(* CODESYS project TouchPanel-PIO3_MB_EC.ecp

Project tree, tasks and I/O mapping:
  TP_EtherCat : TP600 10.1 1280x800 PIO3 CP , WAGO, order no. 0762-5304, version 5.13.2.32
    application Application
      libraries: ; VisuDialogs, * (System); SysFile23, 3.5.13.0 (System); VisuElemBase, 3.5.13.20 (System); SysPlcCtrl23, 3.5.13.0 (System); SysTime, 3.5.9.0 (System)
      task PLC_Task (cyclic, interval t#10ms, priority 13) calls nothing
      task EtherCAT_Task (cyclic, interval 4 ms, priority 6) calls PLC_PRG
      program PLC_PRG [ST]
      data type typDiagnosticStatusWord
      data type typDSW
      data type typEcDiag
      function block fbSdoRead4 [ST]
      function block fbSdoWrite [ST]
      program prgSdoHandling [ST]
    Serial
      COM1 : COM1, WAGO, version 0.0.0.19
    MODBUS
      MODBUS : MODBUS, WAGO, order no. n/a, version 1.1.1.15
        _internal_1006_0001_Master : MODBUS Master, WAGO, order no. n/a, version 1.1.1.15
    CANbus
    e_Display_Onboard_IO : TP600 Onboard IO, WAGO, version 0.0.1.2
        unmapped channels: _IN, _OUT
    EtherCAT_Master : EtherCAT Master, WAGO, version 3.5.13.21
        settings: NetworkName = 'ethX2'; NetworkName = "ethX2"; SelectNetworkByName = TRUE
      _750_354_000_002_EtherCat_fieldbus_coupler : 750-354/000-002 EtherCat fieldbus coupler, WAGO, order no. 750-354/000-002, version Revision=16#10010002
          settings: ModularDevice = True; MDP_InputOffsets = [0,224,0,32,96,160]; MDP_OutputOffsets = [0,0,224,32,96,160]; Physical Address of the Slave = 1001; Sync.Length = 30; Sync.Length = 30; FMMU.Global Start Address = 16#02000000; FMMU.Length = 30; FMMU.Physical Start Address = 16#1800; FMMU.Access = 16#02; FMMU.Global Start Address = 16#01000000; FMMU.Length = 30; FMMU.Physical Start Address = 16#2400; FMMU.Access = 16#01; FMMU.Global Start Address = 16#00080000; FMMU.Physical Start Address = 16#080D; FMMU.Access = 16#01; Number of RxPDOs of the Slave = 5; Number of TxPDOs of the Slave = 5; DC sync0 cycletime = 4000; DC sync1 cycletime = 4000; Number of SDO = 1; Explicit Device ID (Upper 8 bits).Index = 16#2134; Explicit Device ID (Upper 8 bits).Subindex = 16#00; Explicit Device ID (Upper 8 bits).Value = 0; Explicit Device ID (Upper 8 bits).Size = 8; Explicit Device ID (Upper 8 bits).AbortIfError = FALSE; Explicit Device ID (Upper 8 bits).JumpToLine = FALSE; Explicit Device ID (Upper 8 bits).Line = 0; Explicit Device ID (Upper 8 bits).CompleteAccess = False; RxTxPdo.NumberofExcludes = 0; RxTxPdo.NumberofEntries = 6; RxTxPdo.Index = 16#16FF; RxTxPdo.Fixed = True; RxTxPdo.Mandatory = True; RxTxPdo.Virtual = False; RxTxPdo.Sm = 2; RxTxPdo.Su = 2; RxTxPdo.Name = 'Output'; RxTxPdo.DependOnSlot = False;
            RxTxPdo.DependOnSlotGroup = False; RxTxPdo.OverwrittenByModule = False; FC Control, K-Bus Cycle Overrun Flag Disable.Index = 16#F200; FC Control, K-Bus Cycle Overrun Flag Disable.SubIndex = 1; FC Control, K-Bus Cycle Overrun Flag Disable.Size = 1; FC Control, K-Bus Cycle Overrun Flag Disable.Offset = 0; FC Control, K-Bus Cycle Overrun Flag Disable.DependOnSlot = False; FC Control, K-Bus Cycle Overrun Flag Disable.DependOnSlotGroup = False; FC Control, Input Process Data Hold Request.Index = 16#F200; FC Control, Input Process Data Hold Request.SubIndex = 2; FC Control, Input Process Data Hold Request.Size = 1; FC Control, Input Process Data Hold Request.Offset = 0; FC Control, Input Process Data Hold Request.DependOnSlot = False; FC Control, Input Process Data Hold Request.DependOnSlotGroup = False; FC Control, Output Process Data Hold Request.Index = 16#F200; FC Control, Output Process Data Hold Request.SubIndex = 3; FC Control, Output Process Data Hold Request.Size = 1; FC Control, Output Process Data Hold Request.Offset = 0; FC Control, Output Process Data Hold Request.DependOnSlot = False; FC Control, Output Process Data Hold Request.DependOnSlotGroup = False; FC Control, Output Process Data Clear Request.Index = 16#F200; FC Control, Output Process Data Clear Request.SubIndex = 4; FC Control, Output Process Data Clear Request.Size = 1; FC Control, Output Process Data Clear Request.Offset = 0; FC Control, Output Process Data Clear Request.DependOnSlot = False; FC Control, Output Process Data Clear Request.DependOnSlotGroup = False; Entry.Index = 16#0000; Entry.SubIndex = 0; Entry.Size = 12; Entry.Offset = 0; Entry.DependOnSlot = False; Entry.DependOnSlotGroup = False; Diagnostics Control Word.Index = 16#F200; Diagnostics Control Word.SubIndex = 5; Diagnostics Control Word.Size = 16; Diagnostics Control Word.Offset = 0; Diagnostics Control Word.DependOnSlot = False; Diagnostics Control Word.DependOnSlotGroup = False; RxTxPdo.NumberofExcludes = 0; RxTxPdo.NumberofEntries = 6;
            RxTxPdo.Index = 16#1602; RxTxPdo.Fixed = True; RxTxPdo.Mandatory = True; RxTxPdo.Virtual = False; RxTxPdo.Sm = 2; RxTxPdo.Su = 0; RxTxPdo.Name = 'Output(s)'; RxTxPdo.DependOnSlot = True; RxTxPdo.DependOnSlotGroup = False; RxTxPdo.OverwrittenByModule = True; Channel 1, Control.Index = 16#7020; Channel 1, Control.SubIndex = 1; Channel 1, Control.Size = 8; Channel 1, Control.Offset = 0; Channel 1, Control.DependOnSlot = True; Channel 1, Control.DependOnSlotGroup = True; ---.Index = 16#0000; ---.SubIndex = 0; ---.Size = 8; ---.Offset = 0; ---.DependOnSlot = False; ---.DependOnSlotGroup = False; Channel 1, Word 1.Index = 16#7020; Channel 1, Word 1.SubIndex = 2; Channel 1, Word 1.Size = 16; Channel 1, Word 1.Offset = 0; Channel 1, Word 1.DependOnSlot = True; Channel 1, Word 1.DependOnSlotGroup = True; Channel 2, Control.Index = 16#7020; Channel 2, Control.SubIndex = 3; Channel 2, Control.Size = 8; Channel 2, Control.Offset = 0; Channel 2, Control.DependOnSlot = True; Channel 2, Control.DependOnSlotGroup = True; ---.Index = 16#0000; ---.SubIndex = 0; ---.Size = 8; ---.Offset = 0; ---.DependOnSlot = False; ---.DependOnSlotGroup = False;
            Channel 2, Word 1.Index = 16#7020; Channel 2, Word 1.SubIndex = 4; Channel 2, Word 1.Size = 16; Channel 2, Word 1.Offset = 0; Channel 2, Word 1.DependOnSlot = True; Channel 2, Word 1.DependOnSlotGroup = True; RxTxPdo.NumberofExcludes = 0; RxTxPdo.NumberofEntries = 6; RxTxPdo.Index = 16#1603; RxTxPdo.Fixed = True; RxTxPdo.Mandatory = True; RxTxPdo.Virtual = False; RxTxPdo.Sm = 2; RxTxPdo.Su = 0; RxTxPdo.Name = 'Output(s)'; RxTxPdo.DependOnSlot = True; RxTxPdo.DependOnSlotGroup = False; RxTxPdo.OverwrittenByModule = True; Channel 1, Control.Index = 16#7030; Channel 1, Control.SubIndex = 1; Channel 1, Control.Size = 8; Channel 1, Control.Offset = 0; Channel 1, Control.DependOnSlot = True; Channel 1, Control.DependOnSlotGroup = True; ---.Index = 16#0000; ---.SubIndex = 0; ---.Size = 8; ---.Offset = 0; ---.DependOnSlot = False; ---.DependOnSlotGroup = False; Channel 1, Word 1.Index = 16#7030; Channel 1, Word 1.SubIndex = 2; Channel 1, Word 1.Size = 16; Channel 1, Word 1.Offset = 0; Channel 1, Word 1.DependOnSlot = True; Channel 1, Word 1.DependOnSlotGroup = True; Channel 2, Control.Index = 16#7030; Channel 2, Control.SubIndex = 3; Channel 2, Control.Size = 8; Channel 2, Control.Offset = 0;
            Channel 2, Control.DependOnSlot = True; Channel 2, Control.DependOnSlotGroup = True; ---.Index = 16#0000; ---.SubIndex = 0; ---.Size = 8; ---.Offset = 0; ---.DependOnSlot = False; ---.DependOnSlotGroup = False; Channel 2, Word 1.Index = 16#7030; Channel 2, Word 1.SubIndex = 4; Channel 2, Word 1.Size = 16; Channel 2, Word 1.Offset = 0; Channel 2, Word 1.DependOnSlot = True; Channel 2, Word 1.DependOnSlotGroup = True; RxTxPdo.NumberofExcludes = 0; RxTxPdo.NumberofEntries = 6; RxTxPdo.Index = 16#1604; RxTxPdo.Fixed = True; RxTxPdo.Mandatory = True; RxTxPdo.Virtual = False; RxTxPdo.Sm = 2; RxTxPdo.Su = 0; RxTxPdo.Name = 'Output(s)'; RxTxPdo.DependOnSlot = True; RxTxPdo.DependOnSlotGroup = False; RxTxPdo.OverwrittenByModule = True; Channel 1, Control.Index = 16#7040; Channel 1, Control.SubIndex = 1; Channel 1, Control.Size = 8; Channel 1, Control.Offset = 0; Channel 1, Control.DependOnSlot = True; Channel 1, Control.DependOnSlotGroup = True; ---.Index = 16#0000; ---.SubIndex = 0; ---.Size = 8; ---.Offset = 0; ---.DependOnSlot = False; ---.DependOnSlotGroup = False; Channel 1, Word 1.Index = 16#7040; Channel 1, Word 1.SubIndex = 2;
            Channel 1, Word 1.Size = 16; Channel 1, Word 1.Offset = 0; Channel 1, Word 1.DependOnSlot = True; Channel 1, Word 1.DependOnSlotGroup = True; Channel 2, Control.Index = 16#7040; Channel 2, Control.SubIndex = 3; Channel 2, Control.Size = 8; Channel 2, Control.Offset = 0; Channel 2, Control.DependOnSlot = True; Channel 2, Control.DependOnSlotGroup = True; ---.Index = 16#0000; ---.SubIndex = 0; ---.Size = 8; ---.Offset = 0; ---.DependOnSlot = False; ---.DependOnSlotGroup = False; Channel 2, Word 1.Index = 16#7040; Channel 2, Word 1.SubIndex = 4; Channel 2, Word 1.Size = 16; Channel 2, Word 1.Offset = 0; Channel 2, Word 1.DependOnSlot = True; Channel 2, Word 1.DependOnSlotGroup = True; RxTxPdo.NumberofExcludes = 0; RxTxPdo.NumberofEntries = 16; RxTxPdo.Index = 16#1601; RxTxPdo.Fixed = True; RxTxPdo.Mandatory = True; RxTxPdo.Virtual = False; RxTxPdo.Sm = 2; RxTxPdo.Su = 0; RxTxPdo.Name = 'Output(s)'; RxTxPdo.DependOnSlot = True; RxTxPdo.DependOnSlotGroup = False; RxTxPdo.OverwrittenByModule = True; Channel 1, Data 1.Index = 16#7010; Channel 1, Data 1.SubIndex = 1; Channel 1, Data 1.Size = 1; Channel 1, Data 1.Offset = 0; Channel 1, Data 1.DependOnSlot = True; Channel 1, Data 1.DependOnSlotGroup = True;
            Channel 2, Data 1.Index = 16#7010; Channel 2, Data 1.SubIndex = 2; Channel 2, Data 1.Size = 1; Channel 2, Data 1.Offset = 0; Channel 2, Data 1.DependOnSlot = True; Channel 2, Data 1.DependOnSlotGroup = True; Channel 3, Data 1.Index = 16#7010; Channel 3, Data 1.SubIndex = 3; Channel 3, Data 1.Size = 1; Channel 3, Data 1.Offset = 0; Channel 3, Data 1.DependOnSlot = True; Channel 3, Data 1.DependOnSlotGroup = True; Channel 4, Data 1.Index = 16#7010; Channel 4, Data 1.SubIndex = 4; Channel 4, Data 1.Size = 1; Channel 4, Data 1.Offset = 0; Channel 4, Data 1.DependOnSlot = True; Channel 4, Data 1.DependOnSlotGroup = True; Channel 5, Data 1.Index = 16#7010; Channel 5, Data 1.SubIndex = 5; Channel 5, Data 1.Size = 1; Channel 5, Data 1.Offset = 0; Channel 5, Data 1.DependOnSlot = True; Channel 5, Data 1.DependOnSlotGroup = True; Channel 6, Data 1.Index = 16#7010; Channel 6, Data 1.SubIndex = 6; Channel 6, Data 1.Size = 1; Channel 6, Data 1.Offset = 0; Channel 6, Data 1.DependOnSlot = True; Channel 6, Data 1.DependOnSlotGroup = True; Channel 7, Data 1.Index = 16#7010; Channel 7, Data 1.SubIndex = 7; Channel 7, Data 1.Size = 1; Channel 7, Data 1.Offset = 0; Channel 7, Data 1.DependOnSlot = True; Channel 7, Data 1.DependOnSlotGroup = True; Channel 8, Data 1.Index = 16#7010; Channel 8, Data 1.SubIndex = 8; Channel 8, Data 1.Size = 1; Channel 8, Data 1.Offset = 0;
            Channel 8, Data 1.DependOnSlot = True; Channel 8, Data 1.DependOnSlotGroup = True; Channel 9, Data 1.Index = 16#7010; Channel 9, Data 1.SubIndex = 9; Channel 9, Data 1.Size = 1; Channel 9, Data 1.Offset = 0; Channel 9, Data 1.DependOnSlot = True; Channel 9, Data 1.DependOnSlotGroup = True; Channel 10, Data 1.Index = 16#7010; Channel 10, Data 1.SubIndex = 10; Channel 10, Data 1.Size = 1; Channel 10, Data 1.Offset = 0; Channel 10, Data 1.DependOnSlot = True; Channel 10, Data 1.DependOnSlotGroup = True; Channel 11, Data 1.Index = 16#7010; Channel 11, Data 1.SubIndex = 11; Channel 11, Data 1.Size = 1; Channel 11, Data 1.Offset = 0; Channel 11, Data 1.DependOnSlot = True; Channel 11, Data 1.DependOnSlotGroup = True; Channel 12, Data 1.Index = 16#7010; Channel 12, Data 1.SubIndex = 12; Channel 12, Data 1.Size = 1; Channel 12, Data 1.Offset = 0; Channel 12, Data 1.DependOnSlot = True; Channel 12, Data 1.DependOnSlotGroup = True; Channel 13, Data 1.Index = 16#7010; Channel 13, Data 1.SubIndex = 13; Channel 13, Data 1.Size = 1; Channel 13, Data 1.Offset = 0; Channel 13, Data 1.DependOnSlot = True; Channel 13, Data 1.DependOnSlotGroup = True; Channel 14, Data 1.Index = 16#7010; Channel 14, Data 1.SubIndex = 14; Channel 14, Data 1.Size = 1; Channel 14, Data 1.Offset = 0; Channel 14, Data 1.DependOnSlot = True; Channel 14, Data 1.DependOnSlotGroup = True; Channel 15, Data 1.Index = 16#7010; Channel 15, Data 1.SubIndex = 15;
            Channel 15, Data 1.Size = 1; Channel 15, Data 1.Offset = 0; Channel 15, Data 1.DependOnSlot = True; Channel 15, Data 1.DependOnSlotGroup = True; Channel 16, Data 1.Index = 16#7010; Channel 16, Data 1.SubIndex = 16; Channel 16, Data 1.Size = 1; Channel 16, Data 1.Offset = 0; Channel 16, Data 1.DependOnSlot = True; Channel 16, Data 1.DependOnSlotGroup = True; RxTxPdo.NumberofExcludes = 0; RxTxPdo.NumberofEntries = 7; RxTxPdo.Index = 16#1AFF; RxTxPdo.Fixed = True; RxTxPdo.Mandatory = True; RxTxPdo.Virtual = False; RxTxPdo.Sm = 3; RxTxPdo.Su = 3; RxTxPdo.Name = 'Input'; RxTxPdo.DependOnSlot = False; RxTxPdo.DependOnSlotGroup = False; RxTxPdo.OverwrittenByModule = False; FC Status, K-Bus Cycle Overrun Flag.Index = 16#F100; FC Status, K-Bus Cycle Overrun Flag.SubIndex = 1; FC Status, K-Bus Cycle Overrun Flag.Size = 1; FC Status, K-Bus Cycle Overrun Flag.Offset = 0; FC Status, K-Bus Cycle Overrun Flag.DependOnSlot = False; FC Status, K-Bus Cycle Overrun Flag.DependOnSlotGroup = False; FC Status, Input Process Data Hold Ack..Index = 16#F100; FC Status, Input Process Data Hold Ack..SubIndex = 2; FC Status, Input Process Data Hold Ack..Size = 1; FC Status, Input Process Data Hold Ack..Offset = 0; FC Status, Input Process Data Hold Ack..DependOnSlot = False; FC Status, Input Process Data Hold Ack..DependOnSlotGroup = False; FC Status, Output Process Data Hold Ack..Index = 16#F100; FC Status, Output Process Data Hold Ack..SubIndex = 3; FC Status, Output Process Data Hold Ack..Size = 1; FC Status, Output Process Data Hold Ack..Offset = 0; FC Status, Output Process Data Hold Ack..DependOnSlot = False; FC Status, Output Process Data Hold Ack..DependOnSlotGroup = False;
            FC Status, Output Process Data Clear Ack..Index = 16#F100; FC Status, Output Process Data Clear Ack..SubIndex = 4; FC Status, Output Process Data Clear Ack..Size = 1; FC Status, Output Process Data Clear Ack..Offset = 0; FC Status, Output Process Data Clear Ack..DependOnSlot = False; FC Status, Output Process Data Clear Ack..DependOnSlotGroup = False; Entry.Index = 16#0000; Entry.SubIndex = 0; Entry.Size = 11; Entry.Offset = 0; Entry.DependOnSlot = False; Entry.DependOnSlotGroup = False; Diagnosis History, New Message Available.Index = 16#10F3; Diagnosis History, New Message Available.SubIndex = 4; Diagnosis History, New Message Available.Size = 1; Diagnosis History, New Message Available.Offset = 0; Diagnosis History, New Message Available.DependOnSlot = False; Diagnosis History, New Message Available.DependOnSlotGroup = False; Diagnostics Status Word.Index = 16#F100; Diagnostics Status Word.SubIndex = 5; Diagnostics Status Word.Size = 16; Diagnostics Status Word.Offset = 0; Diagnostics Status Word.DependOnSlot = False; Diagnostics Status Word.DependOnSlotGroup = False; RxTxPdo.NumberofExcludes = 0; RxTxPdo.NumberofEntries = 6; RxTxPdo.Index = 16#1A02; RxTxPdo.Fixed = True; RxTxPdo.Mandatory = True; RxTxPdo.Virtual = False; RxTxPdo.Sm = 3; RxTxPdo.Su = 0; RxTxPdo.Name = 'Input(s)'; RxTxPdo.DependOnSlot = True; RxTxPdo.DependOnSlotGroup = False; RxTxPdo.OverwrittenByModule = True; Channel 1, Status.Index = 16#6020; Channel 1, Status.SubIndex = 1; Channel 1, Status.Size = 8; Channel 1, Status.Offset = 0;
            Channel 1, Status.DependOnSlot = True; Channel 1, Status.DependOnSlotGroup = True; ---.Index = 16#0000; ---.SubIndex = 0; ---.Size = 8; ---.Offset = 0; ---.DependOnSlot = False; ---.DependOnSlotGroup = False; Channel 1, Word 1.Index = 16#6020; Channel 1, Word 1.SubIndex = 2; Channel 1, Word 1.Size = 16; Channel 1, Word 1.Offset = 0; Channel 1, Word 1.DependOnSlot = True; Channel 1, Word 1.DependOnSlotGroup = True; Channel 2, Status.Index = 16#6020; Channel 2, Status.SubIndex = 3; Channel 2, Status.Size = 8; Channel 2, Status.Offset = 0; Channel 2, Status.DependOnSlot = True; Channel 2, Status.DependOnSlotGroup = True; ---.Index = 16#0000; ---.SubIndex = 0; ---.Size = 8; ---.Offset = 0; ---.DependOnSlot = False; ---.DependOnSlotGroup = False; Channel 2, Word 1.Index = 16#6020; Channel 2, Word 1.SubIndex = 4; Channel 2, Word 1.Size = 16; Channel 2, Word 1.Offset = 0; Channel 2, Word 1.DependOnSlot = True; Channel 2, Word 1.DependOnSlotGroup = True; RxTxPdo.NumberofExcludes = 0; RxTxPdo.NumberofEntries = 6; RxTxPdo.Index = 16#1A03; RxTxPdo.Fixed = True; RxTxPdo.Mandatory = True; RxTxPdo.Virtual = False; RxTxPdo.Sm = 3; RxTxPdo.Su = 0;
            RxTxPdo.Name = 'Input(s)'; RxTxPdo.DependOnSlot = True; RxTxPdo.DependOnSlotGroup = False; RxTxPdo.OverwrittenByModule = True; Channel 1, Status.Index = 16#6030; Channel 1, Status.SubIndex = 1; Channel 1, Status.Size = 8; Channel 1, Status.Offset = 0; Channel 1, Status.DependOnSlot = True; Channel 1, Status.DependOnSlotGroup = True; ---.Index = 16#0000; ---.SubIndex = 0; ---.Size = 8; ---.Offset = 0; ---.DependOnSlot = False; ---.DependOnSlotGroup = False; Channel 1, Word 1.Index = 16#6030; Channel 1, Word 1.SubIndex = 2; Channel 1, Word 1.Size = 16; Channel 1, Word 1.Offset = 0; Channel 1, Word 1.DependOnSlot = True; Channel 1, Word 1.DependOnSlotGroup = True; Channel 2, Status.Index = 16#6030; Channel 2, Status.SubIndex = 3; Channel 2, Status.Size = 8; Channel 2, Status.Offset = 0; Channel 2, Status.DependOnSlot = True; Channel 2, Status.DependOnSlotGroup = True; ---.Index = 16#0000; ---.SubIndex = 0; ---.Size = 8; ---.Offset = 0; ---.DependOnSlot = False; ---.DependOnSlotGroup = False; Channel 2, Word 1.Index = 16#6030; Channel 2, Word 1.SubIndex = 4; Channel 2, Word 1.Size = 16; Channel 2, Word 1.Offset = 0; Channel 2, Word 1.DependOnSlot = True; Channel 2, Word 1.DependOnSlotGroup = True;
            RxTxPdo.NumberofExcludes = 0; RxTxPdo.NumberofEntries = 6; RxTxPdo.Index = 16#1A04; RxTxPdo.Fixed = True; RxTxPdo.Mandatory = True; RxTxPdo.Virtual = False; RxTxPdo.Sm = 3; RxTxPdo.Su = 0; RxTxPdo.Name = 'Input(s)'; RxTxPdo.DependOnSlot = True; RxTxPdo.DependOnSlotGroup = False; RxTxPdo.OverwrittenByModule = True; Channel 1, Status.Index = 16#6040; Channel 1, Status.SubIndex = 1; Channel 1, Status.Size = 8; Channel 1, Status.Offset = 0; Channel 1, Status.DependOnSlot = True; Channel 1, Status.DependOnSlotGroup = True; ---.Index = 16#0000; ---.SubIndex = 0; ---.Size = 8; ---.Offset = 0; ---.DependOnSlot = False; ---.DependOnSlotGroup = False; Channel 1, Word 1.Index = 16#6040; Channel 1, Word 1.SubIndex = 2; Channel 1, Word 1.Size = 16; Channel 1, Word 1.Offset = 0; Channel 1, Word 1.DependOnSlot = True; Channel 1, Word 1.DependOnSlotGroup = True; Channel 2, Status.Index = 16#6040; Channel 2, Status.SubIndex = 3; Channel 2, Status.Size = 8; Channel 2, Status.Offset = 0; Channel 2, Status.DependOnSlot = True; Channel 2, Status.DependOnSlotGroup = True; ---.Index = 16#0000; ---.SubIndex = 0; ---.Size = 8; ---.Offset = 0;
            ---.DependOnSlot = False; ---.DependOnSlotGroup = False; Channel 2, Word 1.Index = 16#6040; Channel 2, Word 1.SubIndex = 4; Channel 2, Word 1.Size = 16; Channel 2, Word 1.Offset = 0; Channel 2, Word 1.DependOnSlot = True; Channel 2, Word 1.DependOnSlotGroup = True; RxTxPdo.NumberofExcludes = 0; RxTxPdo.NumberofEntries = 16; RxTxPdo.Index = 16#1A00; RxTxPdo.Fixed = True; RxTxPdo.Mandatory = True; RxTxPdo.Virtual = False; RxTxPdo.Sm = 3; RxTxPdo.Su = 0; RxTxPdo.Name = 'Input(s)'; RxTxPdo.DependOnSlot = True; RxTxPdo.DependOnSlotGroup = False; RxTxPdo.OverwrittenByModule = True; Channel 1, Data 1.Index = 16#6000; Channel 1, Data 1.SubIndex = 1; Channel 1, Data 1.Size = 1; Channel 1, Data 1.Offset = 0; Channel 1, Data 1.DependOnSlot = True; Channel 1, Data 1.DependOnSlotGroup = True; Channel 2, Data 1.Index = 16#6000; Channel 2, Data 1.SubIndex = 2; Channel 2, Data 1.Size = 1; Channel 2, Data 1.Offset = 0; Channel 2, Data 1.DependOnSlot = True; Channel 2, Data 1.DependOnSlotGroup = True; Channel 3, Data 1.Index = 16#6000; Channel 3, Data 1.SubIndex = 3; Channel 3, Data 1.Size = 1; Channel 3, Data 1.Offset = 0; Channel 3, Data 1.DependOnSlot = True; Channel 3, Data 1.DependOnSlotGroup = True; Channel 4, Data 1.Index = 16#6000; Channel 4, Data 1.SubIndex = 4;
            Channel 4, Data 1.Size = 1; Channel 4, Data 1.Offset = 0; Channel 4, Data 1.DependOnSlot = True; Channel 4, Data 1.DependOnSlotGroup = True; Channel 5, Data 1.Index = 16#6000; Channel 5, Data 1.SubIndex = 5; Channel 5, Data 1.Size = 1; Channel 5, Data 1.Offset = 0; Channel 5, Data 1.DependOnSlot = True; Channel 5, Data 1.DependOnSlotGroup = True; Channel 6, Data 1.Index = 16#6000; Channel 6, Data 1.SubIndex = 6; Channel 6, Data 1.Size = 1; Channel 6, Data 1.Offset = 0; Channel 6, Data 1.DependOnSlot = True; Channel 6, Data 1.DependOnSlotGroup = True; Channel 7, Data 1.Index = 16#6000; Channel 7, Data 1.SubIndex = 7; Channel 7, Data 1.Size = 1; Channel 7, Data 1.Offset = 0; Channel 7, Data 1.DependOnSlot = True; Channel 7, Data 1.DependOnSlotGroup = True; Channel 8, Data 1.Index = 16#6000; Channel 8, Data 1.SubIndex = 8; Channel 8, Data 1.Size = 1; Channel 8, Data 1.Offset = 0; Channel 8, Data 1.DependOnSlot = True; Channel 8, Data 1.DependOnSlotGroup = True; Channel 9, Data 1.Index = 16#6000; Channel 9, Data 1.SubIndex = 9; Channel 9, Data 1.Size = 1; Channel 9, Data 1.Offset = 0; Channel 9, Data 1.DependOnSlot = True; Channel 9, Data 1.DependOnSlotGroup = True; Channel 10, Data 1.Index = 16#6000; Channel 10, Data 1.SubIndex = 10; Channel 10, Data 1.Size = 1; Channel 10, Data 1.Offset = 0; Channel 10, Data 1.DependOnSlot = True; Channel 10, Data 1.DependOnSlotGroup = True;
            Channel 11, Data 1.Index = 16#6000; Channel 11, Data 1.SubIndex = 11; Channel 11, Data 1.Size = 1; Channel 11, Data 1.Offset = 0; Channel 11, Data 1.DependOnSlot = True; Channel 11, Data 1.DependOnSlotGroup = True; Channel 12, Data 1.Index = 16#6000; Channel 12, Data 1.SubIndex = 12; Channel 12, Data 1.Size = 1; Channel 12, Data 1.Offset = 0; Channel 12, Data 1.DependOnSlot = True; Channel 12, Data 1.DependOnSlotGroup = True; Channel 13, Data 1.Index = 16#6000; Channel 13, Data 1.SubIndex = 13; Channel 13, Data 1.Size = 1; Channel 13, Data 1.Offset = 0; Channel 13, Data 1.DependOnSlot = True; Channel 13, Data 1.DependOnSlotGroup = True; Channel 14, Data 1.Index = 16#6000; Channel 14, Data 1.SubIndex = 14; Channel 14, Data 1.Size = 1; Channel 14, Data 1.Offset = 0; Channel 14, Data 1.DependOnSlot = True; Channel 14, Data 1.DependOnSlotGroup = True; Channel 15, Data 1.Index = 16#6000; Channel 15, Data 1.SubIndex = 15; Channel 15, Data 1.Size = 1; Channel 15, Data 1.Offset = 0; Channel 15, Data 1.DependOnSlot = True; Channel 15, Data 1.DependOnSlotGroup = True; Channel 16, Data 1.Index = 16#6000; Channel 16, Data 1.SubIndex = 16; Channel 16, Data 1.Size = 1; Channel 16, Data 1.Offset = 0; Channel 16, Data 1.DependOnSlot = True; Channel 16, Data 1.DependOnSlotGroup = True; FC Control, K-Bus Cycle Overrun Flag Disable.Name = 'FC Control, K-Bus Cycle Overrun Flag Disable'; FC Control, K-Bus Cycle Overrun Flag Disable.DataType = 'BIT'; FC Control, K-Bus Cycle Overrun Flag Disable.Default = ''; FC Control, K-Bus Cycle Overrun Flag Disable.Comment = '';
            FC Control, Input Process Data Hold Request.Name = 'FC Control, Input Process Data Hold Request'; FC Control, Input Process Data Hold Request.DataType = 'BIT'; FC Control, Input Process Data Hold Request.Default = ''; FC Control, Input Process Data Hold Request.Comment = ''; FC Control, Output Process Data Hold Request.Name = 'FC Control, Output Process Data Hold Request'; FC Control, Output Process Data Hold Request.DataType = 'BIT'; FC Control, Output Process Data Hold Request.Default = ''; FC Control, Output Process Data Hold Request.Comment = ''; FC Control, Output Process Data Clear Request.Name = 'FC Control, Output Process Data Clear Request'; FC Control, Output Process Data Clear Request.DataType = 'BIT'; FC Control, Output Process Data Clear Request.Default = ''; FC Control, Output Process Data Clear Request.Comment = ''; Entry.Name = ''; Entry.DataType = ''; Entry.Default = ''; Entry.Comment = ''; Diagnostics Control Word.Name = 'Diagnostics Control Word'; Diagnostics Control Word.DataType = 'UINT'; Diagnostics Control Word.Default = ''; Diagnostics Control Word.Comment = ''; Channel 1, Control.Name = 'Channel 1, Control'; Channel 1, Control.DataType = 'USINT'; Channel 1, Control.Default = ''; Channel 1, Control.Comment = ''; ---.Name = '---'; ---.DataType = ''; ---.Default = ''; ---.Comment = ''; Channel 1, Word 1.Name = 'Channel 1, Word 1'; Channel 1, Word 1.DataType = 'UINT'; Channel 1, Word 1.Default = ''; Channel 1, Word 1.Comment = ''; Channel 2, Control.Name = 'Channel 2, Control'; Channel 2, Control.DataType = 'USINT'; Channel 2, Control.Default = ''; Channel 2, Control.Comment = ''; ---.Name = '---'; ---.DataType = ''; ---.Default = ''; ---.Comment = '';
            Channel 2, Word 1.Name = 'Channel 2, Word 1'; Channel 2, Word 1.DataType = 'UINT'; Channel 2, Word 1.Default = ''; Channel 2, Word 1.Comment = ''; Channel 1, Control.Name = 'Channel 1, Control'; Channel 1, Control.DataType = 'USINT'; Channel 1, Control.Default = ''; Channel 1, Control.Comment = ''; ---.Name = '---'; ---.DataType = ''; ---.Default = ''; ---.Comment = ''; Channel 1, Word 1.Name = 'Channel 1, Word 1'; Channel 1, Word 1.DataType = 'UINT'; Channel 1, Word 1.Default = ''; Channel 1, Word 1.Comment = ''; Channel 2, Control.Name = 'Channel 2, Control'; Channel 2, Control.DataType = 'USINT'; Channel 2, Control.Default = ''; Channel 2, Control.Comment = ''; ---.Name = '---'; ---.DataType = ''; ---.Default = ''; ---.Comment = ''; Channel 2, Word 1.Name = 'Channel 2, Word 1'; Channel 2, Word 1.DataType = 'UINT'; Channel 2, Word 1.Default = ''; Channel 2, Word 1.Comment = ''; Channel 1, Control.Name = 'Channel 1, Control'; Channel 1, Control.DataType = 'USINT'; Channel 1, Control.Default = ''; Channel 1, Control.Comment = ''; ---.Name = '---'; ---.DataType = ''; ---.Default = ''; ---.Comment = ''; Channel 1, Word 1.Name = 'Channel 1, Word 1'; Channel 1, Word 1.DataType = 'UINT'; Channel 1, Word 1.Default = ''; Channel 1, Word 1.Comment = '';
            Channel 2, Control.Name = 'Channel 2, Control'; Channel 2, Control.DataType = 'USINT'; Channel 2, Control.Default = ''; Channel 2, Control.Comment = ''; ---.Name = '---'; ---.DataType = ''; ---.Default = ''; ---.Comment = ''; Channel 2, Word 1.Name = 'Channel 2, Word 1'; Channel 2, Word 1.DataType = 'UINT'; Channel 2, Word 1.Default = ''; Channel 2, Word 1.Comment = ''; Channel 1, Data 1.Name = 'Channel 1, Data 1'; Channel 1, Data 1.DataType = 'BOOL'; Channel 1, Data 1.Default = ''; Channel 1, Data 1.Comment = ''; Channel 2, Data 1.Name = 'Channel 2, Data 1'; Channel 2, Data 1.DataType = 'BOOL'; Channel 2, Data 1.Default = ''; Channel 2, Data 1.Comment = ''; Channel 3, Data 1.Name = 'Channel 3, Data 1'; Channel 3, Data 1.DataType = 'BOOL'; Channel 3, Data 1.Default = ''; Channel 3, Data 1.Comment = ''; Channel 4, Data 1.Name = 'Channel 4, Data 1'; Channel 4, Data 1.DataType = 'BOOL'; Channel 4, Data 1.Default = ''; Channel 4, Data 1.Comment = ''; Channel 5, Data 1.Name = 'Channel 5, Data 1'; Channel 5, Data 1.DataType = 'BOOL'; Channel 5, Data 1.Default = ''; Channel 5, Data 1.Comment = ''; Channel 6, Data 1.Name = 'Channel 6, Data 1'; Channel 6, Data 1.DataType = 'BOOL'; Channel 6, Data 1.Default = ''; Channel 6, Data 1.Comment = ''; Channel 7, Data 1.Name = 'Channel 7, Data 1'; Channel 7, Data 1.DataType = 'BOOL'; Channel 7, Data 1.Default = ''; Channel 7, Data 1.Comment = '';
            Channel 8, Data 1.Name = 'Channel 8, Data 1'; Channel 8, Data 1.DataType = 'BOOL'; Channel 8, Data 1.Default = ''; Channel 8, Data 1.Comment = ''; Channel 9, Data 1.Name = 'Channel 9, Data 1'; Channel 9, Data 1.DataType = 'BOOL'; Channel 9, Data 1.Default = ''; Channel 9, Data 1.Comment = ''; Channel 10, Data 1.Name = 'Channel 10, Data 1'; Channel 10, Data 1.DataType = 'BOOL'; Channel 10, Data 1.Default = ''; Channel 10, Data 1.Comment = ''; Channel 11, Data 1.Name = 'Channel 11, Data 1'; Channel 11, Data 1.DataType = 'BOOL'; Channel 11, Data 1.Default = ''; Channel 11, Data 1.Comment = ''; Channel 12, Data 1.Name = 'Channel 12, Data 1'; Channel 12, Data 1.DataType = 'BOOL'; Channel 12, Data 1.Default = ''; Channel 12, Data 1.Comment = ''; Channel 13, Data 1.Name = 'Channel 13, Data 1'; Channel 13, Data 1.DataType = 'BOOL'; Channel 13, Data 1.Default = ''; Channel 13, Data 1.Comment = ''; Channel 14, Data 1.Name = 'Channel 14, Data 1'; Channel 14, Data 1.DataType = 'BOOL'; Channel 14, Data 1.Default = ''; Channel 14, Data 1.Comment = ''; Channel 15, Data 1.Name = 'Channel 15, Data 1'; Channel 15, Data 1.DataType = 'BOOL'; Channel 15, Data 1.Default = ''; Channel 15, Data 1.Comment = ''; Channel 16, Data 1.Name = 'Channel 16, Data 1'; Channel 16, Data 1.DataType = 'BOOL'; Channel 16, Data 1.Default = ''; Channel 16, Data 1.Comment = ''; FC Status, K-Bus Cycle Overrun Flag.Name = 'FC Status, K-Bus Cycle Overrun Flag'; FC Status, K-Bus Cycle Overrun Flag.DataType = 'BIT'; FC Status, K-Bus Cycle Overrun Flag.Default = ''; FC Status, K-Bus Cycle Overrun Flag.Comment = '';
            FC Status, Input Process Data Hold Ack..Name = 'FC Status, Input Process Data Hold Ack.'; FC Status, Input Process Data Hold Ack..DataType = 'BIT'; FC Status, Input Process Data Hold Ack..Default = ''; FC Status, Input Process Data Hold Ack..Comment = ''; FC Status, Output Process Data Hold Ack..Name = 'FC Status, Output Process Data Hold Ack.'; FC Status, Output Process Data Hold Ack..DataType = 'BIT'; FC Status, Output Process Data Hold Ack..Default = ''; FC Status, Output Process Data Hold Ack..Comment = ''; FC Status, Output Process Data Clear Ack..Name = 'FC Status, Output Process Data Clear Ack.'; FC Status, Output Process Data Clear Ack..DataType = 'BIT'; FC Status, Output Process Data Clear Ack..Default = ''; FC Status, Output Process Data Clear Ack..Comment = ''; Entry.Name = ''; Entry.DataType = ''; Entry.Default = ''; Entry.Comment = ''; Diagnosis History, New Message Available.Name = 'Diagnosis History, New Message Available'; Diagnosis History, New Message Available.DataType = 'BIT'; Diagnosis History, New Message Available.Default = ''; Diagnosis History, New Message Available.Comment = ''; Diagnostics Status Word.Name = 'Diagnostics Status Word'; Diagnostics Status Word.DataType = 'UINT'; Diagnostics Status Word.Default = ''; Diagnostics Status Word.Comment = ''; Channel 1, Status.Name = 'Channel 1, Status'; Channel 1, Status.DataType = 'USINT'; Channel 1, Status.Default = ''; Channel 1, Status.Comment = ''; ---.Name = '---'; ---.DataType = ''; ---.Default = ''; ---.Comment = ''; Channel 1, Word 1.Name = 'Channel 1, Word 1'; Channel 1, Word 1.DataType = 'UINT'; Channel 1, Word 1.Default = ''; Channel 1, Word 1.Comment = ''; Channel 2, Status.Name = 'Channel 2, Status'; Channel 2, Status.DataType = 'USINT'; Channel 2, Status.Default = ''; Channel 2, Status.Comment = '';
            ---.Name = '---'; ---.DataType = ''; ---.Default = ''; ---.Comment = ''; Channel 2, Word 1.Name = 'Channel 2, Word 1'; Channel 2, Word 1.DataType = 'UINT'; Channel 2, Word 1.Default = ''; Channel 2, Word 1.Comment = ''; Channel 1, Status.Name = 'Channel 1, Status'; Channel 1, Status.DataType = 'USINT'; Channel 1, Status.Default = ''; Channel 1, Status.Comment = ''; ---.Name = '---'; ---.DataType = ''; ---.Default = ''; ---.Comment = ''; Channel 1, Word 1.Name = 'Channel 1, Word 1'; Channel 1, Word 1.DataType = 'UINT'; Channel 1, Word 1.Default = ''; Channel 1, Word 1.Comment = ''; Channel 2, Status.Name = 'Channel 2, Status'; Channel 2, Status.DataType = 'USINT'; Channel 2, Status.Default = ''; Channel 2, Status.Comment = ''; ---.Name = '---'; ---.DataType = ''; ---.Default = ''; ---.Comment = ''; Channel 2, Word 1.Name = 'Channel 2, Word 1'; Channel 2, Word 1.DataType = 'UINT'; Channel 2, Word 1.Default = ''; Channel 2, Word 1.Comment = ''; Channel 1, Status.Name = 'Channel 1, Status'; Channel 1, Status.DataType = 'USINT'; Channel 1, Status.Default = ''; Channel 1, Status.Comment = ''; ---.Name = '---'; ---.DataType = ''; ---.Default = ''; ---.Comment = '';
            Channel 1, Word 1.Name = 'Channel 1, Word 1'; Channel 1, Word 1.DataType = 'UINT'; Channel 1, Word 1.Default = ''; Channel 1, Word 1.Comment = ''; Channel 2, Status.Name = 'Channel 2, Status'; Channel 2, Status.DataType = 'USINT'; Channel 2, Status.Default = ''; Channel 2, Status.Comment = ''; ---.Name = '---'; ---.DataType = ''; ---.Default = ''; ---.Comment = ''; Channel 2, Word 1.Name = 'Channel 2, Word 1'; Channel 2, Word 1.DataType = 'UINT'; Channel 2, Word 1.Default = ''; Channel 2, Word 1.Comment = ''; Channel 1, Data 1.Name = 'Channel 1, Data 1'; Channel 1, Data 1.DataType = 'BOOL'; Channel 1, Data 1.Default = ''; Channel 1, Data 1.Comment = ''; Channel 2, Data 1.Name = 'Channel 2, Data 1'; Channel 2, Data 1.DataType = 'BOOL'; Channel 2, Data 1.Default = ''; Channel 2, Data 1.Comment = ''; Channel 3, Data 1.Name = 'Channel 3, Data 1'; Channel 3, Data 1.DataType = 'BOOL'; Channel 3, Data 1.Default = ''; Channel 3, Data 1.Comment = ''; Channel 4, Data 1.Name = 'Channel 4, Data 1'; Channel 4, Data 1.DataType = 'BOOL'; Channel 4, Data 1.Default = ''; Channel 4, Data 1.Comment = ''; Channel 5, Data 1.Name = 'Channel 5, Data 1'; Channel 5, Data 1.DataType = 'BOOL'; Channel 5, Data 1.Default = ''; Channel 5, Data 1.Comment = ''; Channel 6, Data 1.Name = 'Channel 6, Data 1'; Channel 6, Data 1.DataType = 'BOOL'; Channel 6, Data 1.Default = ''; Channel 6, Data 1.Comment = '';
            Channel 7, Data 1.Name = 'Channel 7, Data 1'; Channel 7, Data 1.DataType = 'BOOL'; Channel 7, Data 1.Default = ''; Channel 7, Data 1.Comment = ''; Channel 8, Data 1.Name = 'Channel 8, Data 1'; Channel 8, Data 1.DataType = 'BOOL'; Channel 8, Data 1.Default = ''; Channel 8, Data 1.Comment = ''; Channel 9, Data 1.Name = 'Channel 9, Data 1'; Channel 9, Data 1.DataType = 'BOOL'; Channel 9, Data 1.Default = ''; Channel 9, Data 1.Comment = ''; Channel 10, Data 1.Name = 'Channel 10, Data 1'; Channel 10, Data 1.DataType = 'BOOL'; Channel 10, Data 1.Default = ''; Channel 10, Data 1.Comment = ''; Channel 11, Data 1.Name = 'Channel 11, Data 1'; Channel 11, Data 1.DataType = 'BOOL'; Channel 11, Data 1.Default = ''; Channel 11, Data 1.Comment = ''; Channel 12, Data 1.Name = 'Channel 12, Data 1'; Channel 12, Data 1.DataType = 'BOOL'; Channel 12, Data 1.Default = ''; Channel 12, Data 1.Comment = ''; Channel 13, Data 1.Name = 'Channel 13, Data 1'; Channel 13, Data 1.DataType = 'BOOL'; Channel 13, Data 1.Default = ''; Channel 13, Data 1.Comment = ''; Channel 14, Data 1.Name = 'Channel 14, Data 1'; Channel 14, Data 1.DataType = 'BOOL'; Channel 14, Data 1.Default = ''; Channel 14, Data 1.Comment = ''; Channel 15, Data 1.Name = 'Channel 15, Data 1'; Channel 15, Data 1.DataType = 'BOOL'; Channel 15, Data 1.Default = ''; Channel 15, Data 1.Comment = ''; Channel 16, Data 1.Name = 'Channel 16, Data 1'; Channel 16, Data 1.DataType = 'BOOL'; Channel 16, Data 1.Default = ''; Channel 16, Data 1.Comment = ''
          output xDiag01 : BIT  // FC Control, K-Bus Cycle Overrun Flag Disable
          output xDiag02 : BIT  // FC Control, Input Process Data Hold Request
          output xDiag03 : BIT  // FC Control, Output Process Data Hold Request
          output xDiag04 : BIT  // FC Control, Output Process Data Clear Request
          output uiDiag05 : UINT  // Diagnostics Control Word
          input  xDiag06 : BIT  // FC Status, K-Bus Cycle Overrun Flag
          input  xDiag07 : BIT  // FC Status, Input Process Data Hold Ack.
          input  xDiag08 : BIT  // FC Status, Output Process Data Hold Ack.
          input  xDiag09 : BIT  // FC Status, Output Process Data Clear Ack.
          input  xDiag10 : BIT  // Diagnosis History, New Message Available
          input  uiDiag11 : UINT  // Diagnostics Status Word
          unmapped channels: , , , , , , , , , , , , , , , , , , , , , , 
        _750_469_6B_in_ : 750-469 (6B in), WAGO, order no. 750-469 (6B in), version 0
            settings: Number of Outputs = 6; Number of Inputs = 6; Number of Infos about Outputs = 6; Number of Infos about Inputs = 6; RxTxPdo.Virtual = False; RxTxPdo.DependOnSlot = True; RxTxPdo.DependOnSlotGroup = False; RxTxPdo.OverwrittenByModule = True; Channel 1, Control.Offset = 0; Channel 1, Control.DependOnSlot = True; Channel 1, Control.DependOnSlotGroup = True; ---.Index = 16#0000; ---.SubIndex = 0; ---.Size = 8; ---.Offset = 0; ---.DependOnSlot = False; ---.DependOnSlotGroup = False; Channel 1, Word 1.Offset = 0; Channel 1, Word 1.DependOnSlot = True; Channel 1, Word 1.DependOnSlotGroup = True; Channel 2, Control.Offset = 0; Channel 2, Control.DependOnSlot = True; Channel 2, Control.DependOnSlotGroup = True; ---.Index = 16#0000; ---.SubIndex = 0; ---.Size = 8; ---.Offset = 0; ---.DependOnSlot = False; ---.DependOnSlotGroup = False; Channel 2, Word 1.Offset = 0; Channel 2, Word 1.DependOnSlot = True; Channel 2, Word 1.DependOnSlotGroup = True; RxTxPdo.Virtual = False; RxTxPdo.DependOnSlot = True; RxTxPdo.DependOnSlotGroup = False; RxTxPdo.OverwrittenByModule = True; Channel 1, Status.Offset = 0; Channel 1, Status.DependOnSlot = True; Channel 1, Status.DependOnSlotGroup = True; ---.Index = 16#0000;
              ---.SubIndex = 0; ---.Size = 8; ---.Offset = 0; ---.DependOnSlot = False; ---.DependOnSlotGroup = False; Channel 1, Word 1.Offset = 0; Channel 1, Word 1.DependOnSlot = True; Channel 1, Word 1.DependOnSlotGroup = True; Channel 2, Status.Offset = 0; Channel 2, Status.DependOnSlot = True; Channel 2, Status.DependOnSlotGroup = True; ---.Index = 16#0000; ---.SubIndex = 0; ---.Size = 8; ---.Offset = 0; ---.DependOnSlot = False; ---.DependOnSlotGroup = False; Channel 2, Word 1.Offset = 0; Channel 2, Word 1.DependOnSlot = True; Channel 2, Word 1.DependOnSlotGroup = True; Channel 1, Control.Default = ''; ---.Name = '---'; ---.DataType = ''; ---.Default = ''; ---.Comment = ''; Channel 1, Word 1.Default = ''; Channel 2, Control.Default = ''; ---.Name = '---'; ---.DataType = ''; ---.Default = ''; ---.Comment = ''; Channel 2, Word 1.Default = ''; Channel 1, Status.Default = ''; ---.Name = '---'; ---.DataType = ''; ---.Default = ''; ---.Comment = ''; Channel 1, Word 1.Default = ''; Channel 2, Status.Default = ''; ---.Name = '---';
              ---.DataType = ''; ---.Default = ''; ---.Comment = ''; Channel 2, Word 1.Default = ''
            input  uiTemp01Raw : UINT  // Channel 1, Word 1
            input  usiThermoStatus : USINT  // Channel 2, Status
            input  uiTemp02Raw : UINT  // Channel 2, Word 1
            unmapped channels: Channel 1, Control, ---, Channel 1, Word 1, Channel 2, Control, ---, Channel 2, Word 1, Channel 1, Status, ---, ---
        _750_4xx_750_14xx_16b_in_ : 750-4xx / 750-14xx (16b in), WAGO, order no. 750-4xx / 750-14xx (16b in), version 0
            settings: Number of Inputs = 16; Number of Infos about Inputs = 16; RxTxPdo.Virtual = False; RxTxPdo.DependOnSlot = True; RxTxPdo.DependOnSlotGroup = False; RxTxPdo.OverwrittenByModule = True; Channel 1, Data 1.Offset = 0; Channel 1, Data 1.DependOnSlot = True; Channel 1, Data 1.DependOnSlotGroup = True; Channel 2, Data 1.Offset = 0; Channel 2, Data 1.DependOnSlot = True; Channel 2, Data 1.DependOnSlotGroup = True; Channel 3, Data 1.Offset = 0; Channel 3, Data 1.DependOnSlot = True; Channel 3, Data 1.DependOnSlotGroup = True; Channel 4, Data 1.Offset = 0; Channel 4, Data 1.DependOnSlot = True; Channel 4, Data 1.DependOnSlotGroup = True; Channel 5, Data 1.Offset = 0; Channel 5, Data 1.DependOnSlot = True; Channel 5, Data 1.DependOnSlotGroup = True; Channel 6, Data 1.Offset = 0; Channel 6, Data 1.DependOnSlot = True; Channel 6, Data 1.DependOnSlotGroup = True; Channel 7, Data 1.Offset = 0; Channel 7, Data 1.DependOnSlot = True; Channel 7, Data 1.DependOnSlotGroup = True; Channel 8, Data 1.Offset = 0; Channel 8, Data 1.DependOnSlot = True; Channel 8, Data 1.DependOnSlotGroup = True; Channel 9, Data 1.Offset = 0; Channel 9, Data 1.DependOnSlot = True; Channel 9, Data 1.DependOnSlotGroup = True; Channel 10, Data 1.Offset = 0; Channel 10, Data 1.DependOnSlot = True; Channel 10, Data 1.DependOnSlotGroup = True; Channel 11, Data 1.Offset = 0; Channel 11, Data 1.DependOnSlot = True; Channel 11, Data 1.DependOnSlotGroup = True; Channel 12, Data 1.Offset = 0;
              Channel 12, Data 1.DependOnSlot = True; Channel 12, Data 1.DependOnSlotGroup = True; Channel 13, Data 1.Offset = 0; Channel 13, Data 1.DependOnSlot = True; Channel 13, Data 1.DependOnSlotGroup = True; Channel 14, Data 1.Offset = 0; Channel 14, Data 1.DependOnSlot = True; Channel 14, Data 1.DependOnSlotGroup = True; Channel 15, Data 1.Offset = 0; Channel 15, Data 1.DependOnSlot = True; Channel 15, Data 1.DependOnSlotGroup = True; Channel 16, Data 1.Offset = 0; Channel 16, Data 1.DependOnSlot = True; Channel 16, Data 1.DependOnSlotGroup = True; Channel 1, Data 1.Default = ''; Channel 2, Data 1.Default = ''; Channel 3, Data 1.Default = ''; Channel 4, Data 1.Default = ''; Channel 5, Data 1.Default = ''; Channel 6, Data 1.Default = ''; Channel 7, Data 1.Default = ''; Channel 8, Data 1.Default = ''; Channel 9, Data 1.Default = ''; Channel 10, Data 1.Default = ''; Channel 11, Data 1.Default = ''; Channel 12, Data 1.Default = ''; Channel 13, Data 1.Default = ''; Channel 14, Data 1.Default = ''; Channel 15, Data 1.Default = ''; Channel 16, Data 1.Default = ''
            input  xIn01 : BIT  // Channel 1, Data 1
            input  xIn02 : BIT  // Channel 2, Data 1
            input  xIn03 : BIT  // Channel 3, Data 1
            unmapped channels: Channel 4, Data 1, Channel 5, Data 1, Channel 6, Data 1, Channel 7, Data 1, Channel 8, Data 1, Channel 9, Data 1, Channel 10, Data 1, Channel 11, Data 1, Channel 12, Data 1, Channel 13, Data 1, Channel 14, Data 1, Channel 15, Data 1, Channel 16, Data 1
        _750_5xx_750_15xx_16b_out_ : 750-5xx / 750-15xx (16b out), WAGO, order no. 750-5xx / 750-15xx (16b out), version 0
            settings: Number of Outputs = 16; Number of Infos about Outputs = 16; RxTxPdo.Virtual = False; RxTxPdo.DependOnSlot = True; RxTxPdo.DependOnSlotGroup = False; RxTxPdo.OverwrittenByModule = True; Channel 1, Data 1.Offset = 0; Channel 1, Data 1.DependOnSlot = True; Channel 1, Data 1.DependOnSlotGroup = True; Channel 2, Data 1.Offset = 0; Channel 2, Data 1.DependOnSlot = True; Channel 2, Data 1.DependOnSlotGroup = True; Channel 3, Data 1.Offset = 0; Channel 3, Data 1.DependOnSlot = True; Channel 3, Data 1.DependOnSlotGroup = True; Channel 4, Data 1.Offset = 0; Channel 4, Data 1.DependOnSlot = True; Channel 4, Data 1.DependOnSlotGroup = True; Channel 5, Data 1.Offset = 0; Channel 5, Data 1.DependOnSlot = True; Channel 5, Data 1.DependOnSlotGroup = True; Channel 6, Data 1.Offset = 0; Channel 6, Data 1.DependOnSlot = True; Channel 6, Data 1.DependOnSlotGroup = True; Channel 7, Data 1.Offset = 0; Channel 7, Data 1.DependOnSlot = True; Channel 7, Data 1.DependOnSlotGroup = True; Channel 8, Data 1.Offset = 0; Channel 8, Data 1.DependOnSlot = True; Channel 8, Data 1.DependOnSlotGroup = True; Channel 9, Data 1.Offset = 0; Channel 9, Data 1.DependOnSlot = True; Channel 9, Data 1.DependOnSlotGroup = True; Channel 10, Data 1.Offset = 0; Channel 10, Data 1.DependOnSlot = True; Channel 10, Data 1.DependOnSlotGroup = True; Channel 11, Data 1.Offset = 0; Channel 11, Data 1.DependOnSlot = True; Channel 11, Data 1.DependOnSlotGroup = True; Channel 12, Data 1.Offset = 0;
              Channel 12, Data 1.DependOnSlot = True; Channel 12, Data 1.DependOnSlotGroup = True; Channel 13, Data 1.Offset = 0; Channel 13, Data 1.DependOnSlot = True; Channel 13, Data 1.DependOnSlotGroup = True; Channel 14, Data 1.Offset = 0; Channel 14, Data 1.DependOnSlot = True; Channel 14, Data 1.DependOnSlotGroup = True; Channel 15, Data 1.Offset = 0; Channel 15, Data 1.DependOnSlot = True; Channel 15, Data 1.DependOnSlotGroup = True; Channel 16, Data 1.Offset = 0; Channel 16, Data 1.DependOnSlot = True; Channel 16, Data 1.DependOnSlotGroup = True; Channel 1, Data 1.Default = ''; Channel 2, Data 1.Default = ''; Channel 3, Data 1.Default = ''; Channel 4, Data 1.Default = ''; Channel 5, Data 1.Default = ''; Channel 6, Data 1.Default = ''; Channel 7, Data 1.Default = ''; Channel 8, Data 1.Default = ''; Channel 9, Data 1.Default = ''; Channel 10, Data 1.Default = ''; Channel 11, Data 1.Default = ''; Channel 12, Data 1.Default = ''; Channel 13, Data 1.Default = ''; Channel 14, Data 1.Default = ''; Channel 15, Data 1.Default = ''; Channel 16, Data 1.Default = ''
            output xOut1504_01 : BIT  // Channel 1, Data 1
            output xOut1504_02 : BIT  // Channel 2, Data 1
            output xOut1504_03 : BIT  // Channel 3, Data 1
            unmapped channels: Channel 4, Data 1, Channel 5, Data 1, Channel 6, Data 1, Channel 7, Data 1, Channel 8, Data 1, Channel 9, Data 1, Channel 10, Data 1, Channel 11, Data 1, Channel 12, Data 1, Channel 13, Data 1, Channel 14, Data 1, Channel 15, Data 1, Channel 16, Data 1
        _750_467_6B_in_ : 750-467 (6B in), WAGO, order no. 750-467 (6B in), version 0
            settings: Number of Outputs = 6; Number of Inputs = 6; Number of Infos about Outputs = 6; Number of Infos about Inputs = 6; RxTxPdo.Virtual = False; RxTxPdo.DependOnSlot = True; RxTxPdo.DependOnSlotGroup = False; RxTxPdo.OverwrittenByModule = True; Channel 1, Control.Offset = 0; Channel 1, Control.DependOnSlot = True; Channel 1, Control.DependOnSlotGroup = True; ---.Index = 16#0000; ---.SubIndex = 0; ---.Size = 8; ---.Offset = 0; ---.DependOnSlot = False; ---.DependOnSlotGroup = False; Channel 1, Word 1.Offset = 0; Channel 1, Word 1.DependOnSlot = True; Channel 1, Word 1.DependOnSlotGroup = True; Channel 2, Control.Offset = 0; Channel 2, Control.DependOnSlot = True; Channel 2, Control.DependOnSlotGroup = True; ---.Index = 16#0000; ---.SubIndex = 0; ---.Size = 8; ---.Offset = 0; ---.DependOnSlot = False; ---.DependOnSlotGroup = False; Channel 2, Word 1.Offset = 0; Channel 2, Word 1.DependOnSlot = True; Channel 2, Word 1.DependOnSlotGroup = True; RxTxPdo.Virtual = False; RxTxPdo.DependOnSlot = True; RxTxPdo.DependOnSlotGroup = False; RxTxPdo.OverwrittenByModule = True; Channel 1, Status.Offset = 0; Channel 1, Status.DependOnSlot = True; Channel 1, Status.DependOnSlotGroup = True; ---.Index = 16#0000;
              ---.SubIndex = 0; ---.Size = 8; ---.Offset = 0; ---.DependOnSlot = False; ---.DependOnSlotGroup = False; Channel 1, Word 1.Offset = 0; Channel 1, Word 1.DependOnSlot = True; Channel 1, Word 1.DependOnSlotGroup = True; Channel 2, Status.Offset = 0; Channel 2, Status.DependOnSlot = True; Channel 2, Status.DependOnSlotGroup = True; ---.Index = 16#0000; ---.SubIndex = 0; ---.Size = 8; ---.Offset = 0; ---.DependOnSlot = False; ---.DependOnSlotGroup = False; Channel 2, Word 1.Offset = 0; Channel 2, Word 1.DependOnSlot = True; Channel 2, Word 1.DependOnSlotGroup = True; Channel 1, Control.Default = ''; ---.Name = '---'; ---.DataType = ''; ---.Default = ''; ---.Comment = ''; Channel 1, Word 1.Default = ''; Channel 2, Control.Default = ''; ---.Name = '---'; ---.DataType = ''; ---.Default = ''; ---.Comment = ''; Channel 2, Word 1.Default = ''; Channel 1, Status.Default = ''; ---.Name = '---'; ---.DataType = ''; ---.Default = ''; ---.Comment = ''; Channel 1, Word 1.Default = ''; Channel 2, Status.Default = ''; ---.Name = '---';
              ---.DataType = ''; ---.Default = ''; ---.Comment = ''; Channel 2, Word 1.Default = ''
            input  uiAnalog01Raw : UINT  // Channel 1, Word 1
            input  uiAnalog02Raw : UINT  // Channel 2, Word 1
            unmapped channels: Channel 1, Control, ---, Channel 1, Word 1, Channel 2, Control, ---, Channel 2, Word 1, Channel 1, Status, ---, Channel 2, Status, ---
        _750_550_6B_out_ : 750-550 (6B out), WAGO, order no. 750-550 (6B out), version 0
            settings: Number of Outputs = 6; Number of Inputs = 6; Number of Infos about Outputs = 6; Number of Infos about Inputs = 6; RxTxPdo.Virtual = False; RxTxPdo.DependOnSlot = True; RxTxPdo.DependOnSlotGroup = False; RxTxPdo.OverwrittenByModule = True; Channel 1, Control.Offset = 0; Channel 1, Control.DependOnSlot = True; Channel 1, Control.DependOnSlotGroup = True; ---.Index = 16#0000; ---.SubIndex = 0; ---.Size = 8; ---.Offset = 0; ---.DependOnSlot = False; ---.DependOnSlotGroup = False; Channel 1, Word 1.Offset = 0; Channel 1, Word 1.DependOnSlot = True; Channel 1, Word 1.DependOnSlotGroup = True; Channel 2, Control.Offset = 0; Channel 2, Control.DependOnSlot = True; Channel 2, Control.DependOnSlotGroup = True; ---.Index = 16#0000; ---.SubIndex = 0; ---.Size = 8; ---.Offset = 0; ---.DependOnSlot = False; ---.DependOnSlotGroup = False; Channel 2, Word 1.Offset = 0; Channel 2, Word 1.DependOnSlot = True; Channel 2, Word 1.DependOnSlotGroup = True; RxTxPdo.Virtual = False; RxTxPdo.DependOnSlot = True; RxTxPdo.DependOnSlotGroup = False; RxTxPdo.OverwrittenByModule = True; Channel 1, Status.Offset = 0; Channel 1, Status.DependOnSlot = True; Channel 1, Status.DependOnSlotGroup = True; ---.Index = 16#0000;
              ---.SubIndex = 0; ---.Size = 8; ---.Offset = 0; ---.DependOnSlot = False; ---.DependOnSlotGroup = False; Channel 1, Word 1.Offset = 0; Channel 1, Word 1.DependOnSlot = True; Channel 1, Word 1.DependOnSlotGroup = True; Channel 2, Status.Offset = 0; Channel 2, Status.DependOnSlot = True; Channel 2, Status.DependOnSlotGroup = True; ---.Index = 16#0000; ---.SubIndex = 0; ---.Size = 8; ---.Offset = 0; ---.DependOnSlot = False; ---.DependOnSlotGroup = False; Channel 2, Word 1.Offset = 0; Channel 2, Word 1.DependOnSlot = True; Channel 2, Word 1.DependOnSlotGroup = True; Channel 1, Control.Default = ''; ---.Name = '---'; ---.DataType = ''; ---.Default = ''; ---.Comment = ''; Channel 1, Word 1.Default = ''; Channel 2, Control.Default = ''; ---.Name = '---'; ---.DataType = ''; ---.Default = ''; ---.Comment = ''; Channel 2, Word 1.Default = ''; Channel 1, Status.Default = ''; ---.Name = '---'; ---.DataType = ''; ---.Default = ''; ---.Comment = ''; Channel 1, Word 1.Default = ''; Channel 2, Status.Default = ''; ---.Name = '---';
              ---.DataType = ''; ---.Default = ''; ---.Comment = ''; Channel 2, Word 1.Default = ''
            unmapped channels: Channel 1, Control, ---, Channel 1, Word 1, Channel 2, Control, ---, Channel 2, Word 1, Channel 1, Status, ---, Channel 1, Word 1, Channel 2, Status, ---, Channel 2, Word 1
  Controller_ETHERNET_G3_SD : 750-880, WAGO, order no. 0750-0880, version 0.0.0.9
    Kbus : Kbus, WAGO, version 0.0.0.101
      _16_DI_Generic : 075x-16DI, WAGO, order no. 075x-16DI, version 0.0.0.13
          settings: K-BUS Module slot index = 1
          unmapped channels: _IN
      _16_DO_Generic : 075x-16DO, WAGO, order no. 075x-16DO, version 0.0.0.13
          settings: K-BUS Module slot index = 2
          unmapped channels: _OUT
      _2AI_TC_K_Diagn_Adjust : 0750-0469/0003-0000, WAGO, order no. 0750-0469/0003-0000, version 0.0.0.9
          settings: K-BUS Module slot index = 3
          unmapped channels: _IINT 1, _IINT 2
      _2AI_0_10_VDC_SE : 0750-0467, WAGO, order no. 0750-0467, version 0.0.0.9
          settings: K-BUS Module slot index = 4
          unmapped channels: _IW 1, _IW 2
      _2AO_0_10_VDC : 0750-0550, WAGO, order no. 0750-0550, version 0.0.0.9
          settings: K-BUS Module slot index = 5
          unmapped channels: _QW 1, _QW 2
  TP_ModbusMaster : TP600 10.1 1280x800 PIO3 CP , WAGO, order no. 0762-5304, version 5.13.2.32
    application Application
      libraries: 
      task PLC_Task (cyclic, interval t#50ms, priority 15) calls PLC_PRG
      program PLC_PRG [ST]
      MODBUS/
        data type typController_ETHERNET_G3_SD_tcp
      global variables MODBUS
      data type DUT_Union
    MODBUS
      MODBUS : MODBUS, WAGO, order no. n/a, version 1.1.1.15
        _internal_1006_0001_Master : MODBUS Master, WAGO, order no. n/a, version 1.1.1.15
          _internal_1006_0001_IP_1 : MODBUS IP Interface, WAGO, order no. n/a, version 1.1.1.15
              settings: IP settings.Address = '192.168.1.212'
            PFC200_G2_2ETH_RS_tcp : MODBUS Remote Slave, WAGO, order no. n/a, version 1.1.1.15
                settings: Slave address / Unit identifier = 1
          _internal_1006_0001_IP : MODBUS IP Interface, WAGO, order no. n/a, version 1.1.1.15
              settings: IP settings.Address = '192.168.1.80'
            Controller_ETHERNET_G3_SD_tcp : MODBUS Remote Slave, WAGO, order no. n/a, version 1.1.1.15
                settings: Channel100005.Priority = 1; Channel100005.Cycle Time = 200 ms; Channel100005.Read Length = 16 Registers or Coils; ChannelOffset100010 = 0; Channel100025.Priority = 1; Channel100025.Cycle Time = 200 ms; Channel100025.Read Length = 4 Registers or Coils; ChannelOffset100030 = 0; ChannelOffset100050 = 32; Channel100065.Priority = 1; Channel100065.Cycle Time = 200 ms; Channel100065.Read Length = 8 Registers or Coils; ChannelOffset100070 = 0; ChannelOffset100090 = 1; ChannelOffset100110 = 2; ChannelOffset100130 = 3; ChannelOffset100150 = 4; ChannelOffset100170 = 5; ChannelOffset100190 = 6; ChannelOffset100210 = 7; Channel100225.Priority = 1; Channel100225.Cycle Time = 0 ms; Channel100225.Event Mask = 128; Channel100225.Write Address = 513 Registers or Coils; Channel100225.Write Length = 1 Registers or Coils; ChannelOffset100230 = 0; Channel100245.Priority = 1; Channel100245.Cycle Time = 0 ms; Channel100245.Event Mask = 128; Channel100245.Write Address = 512 Registers or Coils; Channel100245.Write Length = 1 Registers or Coils; ChannelOffset100250 = 0; Slave address / Unit identifier = 1
                input  Application.MODBUS.Controller_ETHERNET_G3_SD_tcp.module_dIn_1 : ARRAY[0..1] OF BYTE  // ChannelMapping100020
                input  Application.MODBUS.Controller_ETHERNET_G3_SD_tcp.aIn_1 : INT  // ChannelMapping100040
                input  Application.MODBUS.Controller_ETHERNET_G3_SD_tcp.module_aIn_2 : ARRAY[0..3] OF BYTE  // ChannelMapping100060
                input  Application.MODBUS.Controller_ETHERNET_G3_SD_tcp.dIn_1 : BOOL  // ChannelMapping100080
                input  Application.MODBUS.Controller_ETHERNET_G3_SD_tcp.dIn_2 : BOOL  // ChannelMapping100100
                input  Application.MODBUS.Controller_ETHERNET_G3_SD_tcp.dIn_3 : BOOL  // ChannelMapping100120
                input  Application.MODBUS.Controller_ETHERNET_G3_SD_tcp.dIn_4 : BOOL  // ChannelMapping100140
                input  Application.MODBUS.Controller_ETHERNET_G3_SD_tcp.dIn_5 : BOOL  // ChannelMapping100160
                input  Application.MODBUS.Controller_ETHERNET_G3_SD_tcp.dIn_6 : BOOL  // ChannelMapping100180
                input  Application.MODBUS.Controller_ETHERNET_G3_SD_tcp.dIn_7 : BOOL  // ChannelMapping100200
                input  Application.MODBUS.Controller_ETHERNET_G3_SD_tcp.dIn_8 : BOOL  // ChannelMapping100220
                output Application.MODBUS.Controller_ETHERNET_G3_SD_tcp.dOut_2 : BOOL  // ChannelMapping100240
                output Application.MODBUS.Controller_ETHERNET_G3_SD_tcp.dOut_1 : BOOL  // ChannelMapping100260
    CANbus
    TP600_Onboard_IO : TP600 Onboard IO, WAGO, version 0.0.1.2
        input  xDI_Panel : BOOL  // _IN._IN
        unmapped channels: _IN, _OUT
    Common.PCI
    Serial
      COM1 : COM1, WAGO, version 0.0.0.19
  PFC200_G2_2ETH_RS : 750-8212 PFC200 G2 2ETH RS, WAGO, order no. 0750-8212, version 5.13.2.32
    application Application
      libraries: ; WagoAppMath, 1.1.1.1 (WAGO)
      task PLC_Task (cyclic, interval t#50ms, priority 15) calls PLC_PRG
      program PLC_PRG [ST]
      global variables MODBUS
    Kbus : Kbus, WAGO, version 1.4.0.2
        unmapped channels: K-BUS diagnostics
    MODBUS
      MODBUS : MODBUS, WAGO, order no. n/a, version 1.1.1.15
        LocalDeviceModbus : MODBUS Slave, WAGO, order no. n/a, version 1.1.1.15
            settings: OffsetMap = 0; OffsetMap = 16; OffsetMap = 32; OffsetMap = 64; OffsetMap = 32; OffsetMap = 0
            output Application.PLC_PRG.myInt : INT  // 
            output Application.PLC_PRG.myWord : WORD  // 
            output Application.PLC_PRG.myReal : REAL  // 
            output Application.PLC_PRG.xMyBOOl : BOOL  // 
            input  Application.PLC_PRG.xRxFromMaster : BOOL  // 
            input  Application.PLC_PRG.rSetPointFromMaster : REAL  // 
          TcpSettings : Modbus TCP Slave, WAGO, order no. n/a, version 1.1.1.15
              settings: TCP connection watchdog = 200 10ms
    Common.PCI
    Serial
      COM1 : COM1, WAGO, version 0.0.0.19
  libraries: WagoAppTime, 1.7.3.3 (WAGO); WagoAppPlcModbus, 1.1.2.3 (WAGO); WagoSysFieldbusModule, 1.9.1.2 (WAGO); WagoAppPowerMeasurement, 1.7.1.3 (WAGO); VisuSymbols, 3.5.10.0 (System); WagoVisuIcons, 1.0.1.0 (WAGO)
  30 Visualizations/
    DynVisuElems/
      building/
        sunblind01/
          image pool sunblind01_img
          function block sunblind01FB [ST]
          visualisation sunblind01Visu
      cogwheels/
        cogwheel01/
          image pool cogwheel01_img
          function block cogwheel01FB [ST]
          visualisation cogwheel01Visu
        cogwheel02/
          image pool cogwheel02_img
          function block cogwheel02FB [ST]
          visualisation cogwheel02Visu
        cogwheel03/
          image pool cogwheel03_img
          function block cogwheel03FB [ST]
          visualisation cogwheel03Visu
  text list GlobalTextList
  image pool ImagePool
  function block ProcessorLoad [ST]
  function block UsrList_Log [ST]
  5ce3da45-db07-42e7-a21c-a00fff4ed8f6|myPics\flags\Germany.png
  5ce3da45-db07-42e7-a21c-a00fff4ed8f6|myPics\flags\France.png
  5ce3da45-db07-42e7-a21c-a00fff4ed8f6|myPics\flags\China.png
  5ce3da45-db07-42e7-a21c-a00fff4ed8f6|myPics\haacke_haus_bauhausvilla_0_org.jpg
  5ce3da45-db07-42e7-a21c-a00fff4ed8f6|myPics\flags\Italy.png
  5ce3da45-db07-42e7-a21c-a00fff4ed8f6|myPics\flags\Japan.png
  5ce3da45-db07-42e7-a21c-a00fff4ed8f6|myPics\flags\Russia.png
  5ce3da45-db07-42e7-a21c-a00fff4ed8f6|myPics\flags\Spain.png
  5ce3da45-db07-42e7-a21c-a00fff4ed8f6|myPics\flags\Thailand.png
  5ce3da45-db07-42e7-a21c-a00fff4ed8f6|myPics\flags\UK.png
  5ce3da45-db07-42e7-a21c-a00fff4ed8f6|myPics\LivingRoom.png
  5ce3da45-db07-42e7-a21c-a00fff4ed8f6|VisuPics\cat000.bmp
  5ce3da45-db07-42e7-a21c-a00fff4ed8f6|VisuPics\cat001.bmp
  5ce3da45-db07-42e7-a21c-a00fff4ed8f6|VisuPics\cat002.bmp
  5ce3da45-db07-42e7-a21c-a00fff4ed8f6|VisuPics\cat003.bmp
  5ce3da45-db07-42e7-a21c-a00fff4ed8f6|VisuPics\cat004.bmp
  5ce3da45-db07-42e7-a21c-a00fff4ed8f6|VisuPics\cat005.bmp
  5ce3da45-db07-42e7-a21c-a00fff4ed8f6|VisuPics\cat006.bmp
  5ce3da45-db07-42e7-a21c-a00fff4ed8f6|VisuPics\cat007.bmp
  5ce3da45-db07-42e7-a21c-a00fff4ed8f6|VisuPics\cat000.jpg
  5ce3da45-db07-42e7-a21c-a00fff4ed8f6|VisuPics\cat001.jpg
  5ce3da45-db07-42e7-a21c-a00fff4ed8f6|VisuPics\cat002.jpg
  5ce3da45-db07-42e7-a21c-a00fff4ed8f6|VisuPics\cat003.jpg
  5ce3da45-db07-42e7-a21c-a00fff4ed8f6|VisuPics\cat004.jpg
  5ce3da45-db07-42e7-a21c-a00fff4ed8f6|VisuPics\cat005.jpg
  5ce3da45-db07-42e7-a21c-a00fff4ed8f6|VisuPics\cat006.jpg
  5ce3da45-db07-42e7-a21c-a00fff4ed8f6|VisuPics\cat007.jpg
*)

// TP_ModbusMaster/Application/MODBUS/typController_ETHERNET_G3_SD_tcp
TYPE typController_ETHERNET_G3_SD_tcp:
STRUCT
	dOut_2: BOOL;
	dOut_1: BOOL;
	dIn_1: BOOL;
	module_dIn_1: ARRAY[0..1] OF BYTE;
	dIn_2: BOOL;
	dIn_3: BOOL;
	dIn_4: BOOL;
	dIn_5: BOOL;
	dIn_6: BOOL;
	dIn_7: BOOL;
	dIn_8: BOOL;
	aIn_1: INT;
	module_aIn_2: ARRAY[0..3] OF BYTE;
END_STRUCT
END_TYPE

// TP_ModbusMaster/Application/DUT_Union
TYPE DUT_Union :
UNION
	abmodule_aIn_2: ARRAY[0..3] OF BYTE;
	awmodule_aIn_2: ARRAY[0..1] OF WORD;
END_UNION
END_TYPE

// TP_EtherCat/Application/typDiagnosticStatusWord
TYPE typDiagnosticStatusWord :
UNION
	wData:	WORD;
	stData:	typDSW;
END_UNION
END_TYPE

// TP_EtherCat/Application/typDSW
TYPE typDSW :
STRUCT
	bTRMNLNUM:	BYTE;
	xCHNUM08:	BIT;
	xCHNUM09:	BIT;
	xCHNUM10:	BIT;
	xEVTCODE11:	BIT;
	xEVTCODE12:	BIT;
	xEVTCODE13:	BIT;
	xCLRACK14:	BIT;
	xEVENT15:	BIT;
END_STRUCT
END_TYPE

// TP_EtherCat/Application/typEcDiag
TYPE typEcDiag :
STRUCT
	EccFcControlKBusCycleOverrunFlagDisable:		BOOL;
	EccFcControlInputProcessDataHoldRequest:		BOOL;
	EccFcControlOutputProcessDataHoldRequest:		BOOL;
	EccFcControlOutputProcessDataClearRequest:		BOOL;
	EccDiagnosticsControlWord:						UINT;
	EccFcStatusKBusCycleOverrunFlag:				BOOL;
	EccFcStatusInputProcessDataHoldAcknowledge:		BOOL;
	EccFcStatusOutputProcessDataHoldAcknowledge:	BOOL;
	EccFcStatusOutputProcessDataClearAcknowledge:	BOOL;
	EccDiagnosisHistoryNewMessageAvailable:			BOOL;
	EccDiagnosticsStatusWord:						UINT;
END_STRUCT
END_TYPE

// TP_ModbusMaster/Application/MODBUS
{attribute 'qualified_only'}
VAR_GLOBAL
	
	
	Controller_ETHERNET_G3_SD_tcp: typController_ETHERNET_G3_SD_tcp;
END_VAR

// PFC200_G2_2ETH_RS/Application/MODBUS
{attribute 'qualified_only'}
VAR_GLOBAL
END_VAR

// TP_EtherCat/Application/PLC_PRG
PROGRAM PLC_PRG
VAR
	xInit:			BOOL;
	a, i, j, uiProcessorLoad: UINT;
	b:				UINT := 3;
	rResult:		REAL;
	stEtherCATDiag:	typEcDiag;
	rTemperature, rPotiPercent: REAL;
	tHelper, tDuration: TIME;
	udiSendFrameCount, udiFramesPerSecond, udiLostFrameCount,
	udiTxErrorFrameCount, udiRxErrorFrameCount: UDINT;
	auiDuration:	ARRAY[0..cMaxIdxDuration] OF UINT;
	xResetStatistics: BOOL;
	uDiagnosticStatusWord: typDiagnosticStatusWord;
	usiBusLoad: USINT;
	
END_VAR
VAR CONSTANT
	cMaxIdxDuration: UINT := 99;
END_VAR

// this programme is running
a := a + 1;

// read the single error variables of the etherCAT connection to my struct variable
stEtherCATDiag.EccFcControlKBusCycleOverrunFlagDisable		:= xDiag01;
stEtherCATDiag.EccFcControlInputProcessDataHoldRequest		:= xDiag02;
stEtherCATDiag.EccFcControlOutputProcessDataHoldRequest		:= xDiag03;
stEtherCATDiag.EccFcControlOutputProcessDataClearRequest	:= xDiag04;
stEtherCATDiag.EccDiagnosticsControlWord					:= uiDiag05;
stEtherCATDiag.EccFcStatusKBusCycleOverrunFlag				:= xDiag06;
stEtherCATDiag.EccFcStatusInputProcessDataHoldAcknowledge	:= xDiag07;
stEtherCATDiag.EccFcStatusOutputProcessDataHoldAcknowledge	:= xDiag08;
stEtherCATDiag.EccFcStatusOutputProcessDataClearAcknowledge	:= xDiag09;
stEtherCATDiag.EccDiagnosisHistoryNewMessageAvailable		:= xDiag10;
stEtherCATDiag.EccDiagnosticsStatusWord						:= uiDiag11;
// see the struct uDiagnosticStatusWord.stData for detailed information
uDiagnosticStatusWord.wData									:= uiDiag11;

// set an output of the output module, connected to the etherCAT coupler when its input is set

xOut1504_01 := xIn01;
//xOut512_01	:= xIn01;

// read analogue values of the analogue modules, connected to the etherCAT coupler
rTemperature := uiTemp01Raw * 0.1;
rPotiPercent := uiAnalog01Raw / 327.6;

// set an output when the poti's value is greater than 50 %
//xOut512_02	:= rPotiPercent > 50.0;

// get actual time
tHelper := TIME();
// stress my controller, which simulates an application just by calculating a sine wave
FOR i := 0 TO b DO
	rResult := 50.0 * SIN(i / 30.0) + 1.0;
END_FOR
// calculate the duration of this process
tDuration := TIME() - tHelper;
// memorize the duration in an array
auiDuration[j] := TO_UINT(tDuration);
// increment the array index
j := (j + 1) MOD (cMaxIdxDuration + 1);

// read statistics of etherCAT connection
EtherCAT_Master.GetStatistics(
	udiSendFrameCount	=> udiSendFrameCount,
	udiFramesPerSecond	=> udiFramesPerSecond,
	udiLostFrameCount	=> udiLostFrameCount,
	udiTxErrorCount		=> udiTxErrorFrameCount,
	udiRxErrorCount		=> udiRxErrorFrameCount);

// reset statistics of etherCAT connection
IF xResetStatistics THEN
	EtherCAT_Master.ClearStatistics();
	xResetStatistics := FALSE;
END_IF;

// read processor load
uiProcessorLoad := ProcessorLoad.ProcessorLoad;

// read and write SDOs, never ever forget to query for the xConfigFinished before!!!! 
IF EtherCAT_Master.xConfigFinished THEN
	prgSdoHandling();
END_IF;

END_PROGRAM

// ProcessorLoad
(*
.. figure:: ../../images/wagologo.png
	:align: right
	:alt: WAGO

:Version: 0.0.14.0

:Date: September 6th 2017	
	
	
**Function** 

- functionblock to set Processorload thresholds and the behavior if load is exceeded

.. figure:: ../../images/ProcessorLoad.png
	:align: right
	:alt: WAGO

  

- The Function Block is based on WagoAppProcessorLoad. 

:Author: WAGO/ u010146



+------------------------+---------------+
|Joscat 0.0.14.0          |06.09.2016     |
+------------------------+---------------+
|ProcessorLoad 0.0.14.0 |06.09.2017     |              
+------------------------+---------------+




*)

FUNCTION_BLOCK ProcessorLoad
VAR_INPUT
	usiThreshold1:USINT:=80;
	usiThreshold2:USINT:=90;
	usiIECShare:USINT:=80;
	eOverLoadAction:WagoAppProcessorLoad.WagoTypesProcessorLoad.eOverloadAction:=0;
	eLogLevel:WagoAppProcessorLoad.WagoTypesProcessorLoad.eLogLevel:=0;	
END_VAR
VAR_IN_OUT
	xTriggerSet:BOOL;
END_VAR
VAR_OUTPUT
	usiCurrentThreshold1: USINT;
	usiCurrentThreshold2: USINT;
	usiCurrentIecShare:USINT;
	xThreshold1Exceeded:BOOL;
	xThreshold2Exceeded:BOOL;
	uiCurrentProcessorLoad:UINT;
END_VAR
VAR
	PL01: FbProcessorLoad;
END_VAR



IF xTriggerSet THEN
	PL01.Reinitialize(usiThreshold1:=usiThreshold1,usiThreshold2:=usiThreshold2,usiIECShare:=usiIECShare,eOverloadAction:=eOverLoadAction,eLogLevel:=eLogLevel);
	xTriggerSet:=FALSE;
END_IF

xThreshold1Exceeded:=PL01.IsThreshold1Reached;
xThreshold2Exceeded:=PL01.IsThreshold2Reached;
uiCurrentProcessorLoad:=PL01.ProcessorLoad;
usiCurrentThreshold1:=PL01._usithreshold1;
usiCurrentThreshold2:=PL01._usithreshold2;
usiCurrentIecShare:=PL01._usiIecShare;

END_FUNCTION_BLOCK

// TP_EtherCat/Application/prgSdoHandling
PROGRAM prgSdoHandling
VAR
//	programme is running
	a:					UINT;

//	read SDOs
	fbGenericReadSdo:	fbSdoRead4;
	uiRdDevice:			UINT := 1001;
	wRdIndex:			WORD := 16#7060;		//  Diagnosis History Objects 0x10F3
	bRdSubindex:		BYTE := 2;
	dwRdValue:			DWORD;
	xRdDone, xRdBusy, xRdError: BOOL;
	eRdError:			IoDrvEthercatLib.ETC_CO_ERROR;

//	write SDOs
	xGenericWriteSdo:	BOOL;
	fbGenericWriteSdo:	fbSdoWrite;
	uiWtDevice:			UINT := 1001;
	wWtIndex:			WORD;
	bWtSubindex:		BYTE;
	dwWtValue:			DWORD;
	bWtDataLength:		BYTE;
	xWtDone, xWtBusy, xWtError: BOOL;
	eWtError:			IoDrvEthercatLib.ETC_CO_ERROR;
END_VAR

// programme is running
a := a + 1;
fbGenericReadSdo(
	uiDevice	:= uiRdDevice,
	wIndex		:= wRdIndex,
	bSubindex	:= bRdSubindex,
	dwValue		=> dwRdValue,
	xDone		=> xRdDone,
	xBusy		=> xRdBusy,
	xError		=> xRdError,
	eError		=> eRdError);

// please check before writing if the writing to this index is allowed, see object dictionary
IF xGenericWriteSdo THEN
	fbGenericWriteSdo(
		uiDevice	:= uiWtDevice,
		wIndex		:= wWtIndex,
		bSubindex	:= bWtSubindex,
		dwValue		:= dwWtValue,
		bDataLength	:= bWtDataLength,
		xDone		=> xWtDone,
		xBusy		=> xWtBusy,
		xError		=> xWtError,
		eError		=> eWtError);
	IF fbGenericWriteSdo.xDone OR fbGenericWriteSdo.xError THEN
		xGenericWriteSdo := FALSE;
	END_IF;
END_IF;

END_PROGRAM

// TP_EtherCat/Application/fbSdoRead4
FUNCTION_BLOCK fbSdoRead4
VAR_INPUT
	uiDevice:		UINT;
	wIndex:			WORD;
	bSubindex:		BYTE;
END_VAR
VAR_OUTPUT
	dwValue:		DWORD; 
	xDone, xBusy, xError: BOOL;
	eError:			IoDrvEthercatLib.ETC_CO_ERROR;
END_VAR
VAR
	fbReadSDO:		IoDrvEthercatLib.ETC_CO_SdoRead4;
	iState:			INT := 10;
	udiSDOAbort:	UDINT;
	abData:			ARRAY [1..4] OF BYTE;
	usiDataLength:	USINT;
	pdwValueAdr:	POINTER TO DWORD;
	xAbort, xDone1:	BOOL;
	usiCom:			USINT := 1;
	usiChannel:		USINT := 1;
END_VAR

CASE iState OF
	10:		// start SDO reading
		fbReadSDO(
			xExecute	:= TRUE,
			xAbort		:= xAbort,
			usiCom		:= usiCom,
			uiDevice	:= uiDevice,
			usiChannel	:= usiChannel,
			wIndex		:= wIndex,
			bySubindex	:= bSubindex,
			udiTimeOut	:= 200,
			xDone		=> xDone1,
			xBusy		=> xBusy,
			xError		=> xError,
			eError		=> eError,
			udiSdoAbort	=> udiSDOAbort,
			abyData		=> abData,
			usiDataLength => usiDataLength);
		IF xBusy THEN
			iState := 10;
		END_IF
		IF xError OR xDone1 THEN
			iState := 20;
		END_IF

	20:
		IF xDone1 THEN 
			pdwValueAdr	:= ADR(abData);
			dwValue		:= pdwValueAdr^;
		END_IF
		
		fbReadSDO(
			xExecute	:= FALSE,
			uiDevice	:= uiDevice,
			usiChannel	:= ,
			wIndex		:= wIndex,
			bySubindex	:= bSubindex,
			udiTimeOut	:= 4000,
			xDone		=> xDone,
			xBusy		=> xBusy,
			xError		=> xError,
			eError		=> eError,
			udiSdoAbort	=> udiSDOAbort,
			abyData		=> abData,
			usiDataLength => usiDataLength);
		iState := 10;
END_CASE

END_FUNCTION_BLOCK

// TP_EtherCat/Application/fbSdoWrite
FUNCTION_BLOCK fbSdoWrite
VAR_INPUT
	uiDevice:		UINT;
	wIndex:			WORD;
	bSubindex:		BYTE;
	dwValue:		DWORD;
	bDataLength:	BYTE;
END_VAR
VAR_OUTPUT
	xDone, xBusy, xError: BOOL;
	eError:			IoDrvEthercatLib.ETC_CO_ERROR;
END_VAR
VAR
	iState:			INT := 10;
	udiSDOAbort:	UDINT;
	abData:			ARRAY [1..4] OF BYTE;
	usiDataLength:	USINT;
	dwValueAdr:		POINTER TO BYTE;
	WriteSDO:		IoDrvEthercatLib.ETC_CO_SdoWrite;
	xAbort:			BOOL := FALSE;
	pBuffer:		IoDrvEthercatLib.CAA.PVOID;
	szDataWritten:	__UXINT;
END_VAR


abData[1] := TO_BYTE(SHR(dwValue, 24));
abData[2] := TO_BYTE(SHR(dwValue, 16));
abData[3] := TO_BYTE(SHR(dwValue, 8));
abData[4] := TO_BYTE(SHR(dwValue, 0));

CASE iState OF 
	10: // start SDO writing
		WriteSDO(
			xExecute	:= TRUE,
			xAbort		:= xAbort,
			usiCom		:= 1,
			uiDevice	:= uiDevice,
			usiChannel	:= ,
			wIndex		:= wIndex,
			bySubindex	:= bSubindex,
			udiTimeOut	:= 1000,
			pBuffer		:= ADR(dwValue),
			szSize		:= bDataLength,
			eMode		:= ETC_CO_MODE.ETC_CO_AUTO,
			xDone		=> xDone,
			xBusy		=> xBusy,
			xError		=> xError,
			eError		=> eError,
			udiSdoAbort	=> ,
			szDataWritten => szDataWritten);
		
		IF xBusy THEN
			iState := 10;
		END_IF
		IF xError OR xDone THEN 
			iState := 20;
		END_IF

	20:
		WriteSDO(
			xExecute	:= FALSE,
			xAbort		:= xAbort,
			usiCom		:= 1,
			uiDevice	:= uiDevice,
			usiChannel	:= ,
			wIndex		:= wIndex,
			bySubindex	:= bSubindex,
			udiTimeOut	:= 1000,
			pBuffer		:= ADR(dwValue),
			szSize		:= bDataLength,
			eMode		:= ETC_CO_MODE.ETC_CO_AUTO,
			xDone		=> xDone,
			xBusy		=> xBusy,
			xError		=> xError,
			eError		=> eError,
			udiSdoAbort	=> ,
			szDataWritten => szDataWritten);
		iState := 10;
END_CASE

END_FUNCTION_BLOCK

// TP_ModbusMaster/Application/PLC_PRG
PROGRAM PLC_PRG
VAR
	iRawThermo: REAL;
	xDI_1: BOOL;
	xDI_2: BOOL;
	xDI_3: BOOL;
	xDI_4: BOOL;
	xDI_5: BOOL;
	abAnalogIn: ARRAY [0..3] OF BYTE;
	uCopy:DUT_Union;
	myvalue: BYTE;
	myInput: BYTE;
	xFrom_Panel: BOOL;
	xGo: BOOL := True;
	eErrorCode			: WagoSysModbusDiag.eRemoteSlaveError;
	eChannelErrorCode1	: WagoSysModbusDiag.eChannelError;
	eChannelErrorCode2	: WagoSysModbusDiag.eChannelError;
	eChannelErrorCode3	: WagoSysModbusDiag.eChannelError;
	eChannelErrorCode4: WagoSysModbusDiag.eChannelError;
	eChannelErrorCode5: WagoSysModbusDiag.eChannelError;
	eChannelErrorCode6: WagoSysModbusDiag.eChannelError;
END_VAR

iRawThermo:=MODBUS.Controller_ETHERNET_G3_SD_tcp.aIn_1/10.0;

xDI_1:=MODBUS.Controller_ETHERNET_G3_SD_tcp.dIn_1;
xDI_2:=MODBUS.Controller_ETHERNET_G3_SD_tcp.dIn_2;
xDI_3:=MODBUS.Controller_ETHERNET_G3_SD_tcp.dIn_3;
xDI_4:=MODBUS.Controller_ETHERNET_G3_SD_tcp.dIn_4;
xDI_5:=MODBUS.Controller_ETHERNET_G3_SD_tcp.dIn_5;

abAnalogIn:=MODBUS.Controller_ETHERNET_G3_SD_tcp.module_aIn_2;
uCopy.abmodule_aIn_2:=abAnalogIn;
uCopy.awmodule_aIn_2[0];



myvalue:=myvalue+1;
//IoConfig_Globals_Mapping.bOut_Panel:=myvalue;


MODBUS.Controller_ETHERNET_G3_SD_tcp.dOut_2:=xGo;

MODBUS.Controller_ETHERNET_G3_SD_tcp.dOut_1:=xGo;
eErrorCode:=Controller_ETHERNET_G3_SD_tcp.GetErrorCode();

eChannelErrorCode1:=Controller_ETHERNET_G3_SD_tcp.GetChannelErrorCode(1);
eChannelErrorCode2:=Controller_ETHERNET_G3_SD_tcp.GetChannelErrorCode(2);
eChannelErrorCode3:=Controller_ETHERNET_G3_SD_tcp.GetChannelErrorCode(3);

eChannelErrorCode4:=Controller_ETHERNET_G3_SD_tcp.GetChannelErrorCode(4);
eChannelErrorCode5:=Controller_ETHERNET_G3_SD_tcp.GetChannelErrorCode(5);
eChannelErrorCode6:=Controller_ETHERNET_G3_SD_tcp.GetChannelErrorCode(6);

END_PROGRAM

// PFC200_G2_2ETH_RS/Application/PLC_PRG
PROGRAM PLC_PRG
VAR
	myInt: INT;
	myWord: WORD;
	myReal: REAL;
	xMyBOOl: BOOL;
	xGo: BOOL;
	xRxFromMaster: BOOL;
	rMySetPoint: REAL;
	rSetPointFromMaster: REAL;
END_VAR

myInT:=myInT+1;
myWord:=myWord+1;

myReal:=myReal+3.141;

xMyBOOl:= TO_BOOL(MyInt MOD 2);

xGo:=xRxFromMaster;

rMySetPoint:=rSetPointFromMaster;

END_PROGRAM

// 30 Visualizations/DynVisuElems/building/sunblind01/sunblind01FB
(*
	
**Function Bock for the sunblind01Visu Element** 
Call one FB instance for every sunblind element in the application

- calling the Visu Element the ITF variable sID needs to be replaced with the variable conected to the input sID at the FB
- the variable , which is connected to the FB input xOpen controls the Visu Element


:Author:
WAGO/ u010146

:Version:
0.0.0.1

:Date:
May 25th 2017

+-------------+---------------+
|Version 0.0.1|Johannes Bachem|
+-------------+---------------+
|snblind01FB|               |
+-------------+---------------+



*)





FUNCTION_BLOCK sunblind01FB
VAR_INPUT
	xOpen:BOOL;
END_VAR
VAR_OUTPUT
	sID:STRING;
END_VAR
VAR
END_VAR

IF xOpen THEN
	sID:='rollo_open';
	ELSE
	sID:='rollo_closed';
END_IF

END_FUNCTION_BLOCK

// 30 Visualizations/DynVisuElems/cogwheels/cogwheel01/cogwheel01FB
FUNCTION_BLOCK cogwheel01FB
VAR_INPUT
	
	xEnable: BOOL;
	uiTimeBase: UINT;
END_VAR
VAR_OUTPUT
	sID:STRING;
END_VAR
VAR
	
	i_0_100:BYTE;
	
	
	T1: TOF;
	PT: TIME;
END_VAR

uiTimeBase:=10;
PT:=UINT_TO_TIME(uiTimeBase);


IF xEnable THEN
	T1(IN:=NOT T1.Q , PT:=PT );
IF NOT T1.Q THEN
	i_0_100:=i_0_100+1;
	IF i_0_100 >100 THEN
		i_0_100:=0;
	END_IF
END_IF

END_IF




IF i_0_100 <=8 THEN
	sID:='zahnrad_animation_frame_0001';
ELSIF i_0_100 >8 AND i_0_100 <=17 THEN
	sID:='zahnrad_animation_frame_0002';
ELSIF i_0_100 >17 AND i_0_100 <=25 THEN
	sID:='zahnrad_animation_frame_0003';
ELSIF i_0_100 >25 AND i_0_100 <=33 THEN
	sID:='zahnrad_animation_frame_0004';
ELSIF i_0_100 >33 AND i_0_100 <=42 THEN
	sID:='zahnrad_animation_frame_0005';
ELSIF i_0_100 >42 AND i_0_100 <=50 THEN
	sID:='zahnrad_animation_frame_0006';
ELSIF i_0_100 >50 AND i_0_100 <=58 THEN
	sID:='zahnrad_animation_frame_0007';
ELSIF i_0_100 >58 AND i_0_100 <=67 THEN
	sID:='zahnrad_animation_frame_0008';
ELSIF i_0_100 >67 AND i_0_100 <=75 THEN
	sID:='zahnrad_animation_frame_0009';
ELSIF i_0_100 >75 AND i_0_100 <=83 THEN
	sID:='zahnrad_animation_frame_0010';
ELSIF i_0_100 >83 AND i_0_100 <=92 THEN
	sID:='zahnrad_animation_frame_0011';
ELSIF i_0_100 >92 AND i_0_100 <=100 THEN
	sID:='zahnrad_animation_frame_0012';

END_IF

END_FUNCTION_BLOCK

// 30 Visualizations/DynVisuElems/cogwheels/cogwheel02/cogwheel02FB
FUNCTION_BLOCK cogwheel02FB
VAR_INPUT
	
	xEnable: BOOL;
	uiTimeBase: UINT;
END_VAR
VAR_OUTPUT
	sID:STRING;
END_VAR
VAR
	i_0_100:BYTE;

	T1: TOF;
	PT: TIME;
END_VAR

uiTimeBase:=10;
PT:=UINT_TO_TIME(uiTimeBase);


IF xEnable THEN
	T1(IN:=NOT T1.Q , PT:=PT );
IF NOT T1.Q THEN
	i_0_100:=i_0_100+1;
	IF i_0_100 >100 THEN
		i_0_100:=0;
	END_IF
END_IF

END_IF




IF i_0_100 <=33 THEN
	sID:='zahnrad07_frame_0001';
ELSIF i_0_100 >33 AND i_0_100 <=67 THEN
	sID:='zahnrad07_frame_0002';
ELSIF i_0_100 >67 AND i_0_100 <=100 THEN
	sID:='zahnrad07_frame_0003';
END_IF

END_FUNCTION_BLOCK

// 30 Visualizations/DynVisuElems/cogwheels/cogwheel03/cogwheel03FB
FUNCTION_BLOCK cogwheel03FB
VAR_INPUT
	xEnable: BOOL;
	uiTimeBase: UINT;
END_VAR
	

VAR_OUTPUT
	sID:STRING;
END_VAR
VAR
	i_0_100:BYTE;
	bPos: BYTE;
	T1: TOF;
	PT: TIME;
END_VAR


uiTimeBase:=10;
PT:=UINT_TO_TIME(uiTimeBase);


IF xEnable THEN
	T1(IN:=NOT T1.Q , PT:=PT );
IF NOT T1.Q THEN
	i_0_100:=i_0_100+1;
	IF i_0_100 >100 THEN
		i_0_100:=0;
	END_IF
END_IF

END_IF



IF i_0_100 <=33 THEN
	sID:='silver-two-gear-cogs-animation-8_frame_0001';
ELSIF i_0_100 >33 AND i_0_100 <=67 THEN
	sID:='silver-two-gear-cogs-animation-8_frame_0002';
ELSIF i_0_100 >67 AND i_0_100 <=100 THEN
	sID:='silver-two-gear-cogs-animation-8_frame_0003';
END_IF

END_FUNCTION_BLOCK

// UsrList_Log
FUNCTION_BLOCK UsrList_Log
VAR_INPUT
	
END_VAR
VAR_OUTPUT
	UserList:ARRAY[1..100] OF STRING;
END_VAR
VAR
	myUsrName: STRING;
	
	UsrIdx: INT;
	i: INT;
	UsrIdxLive:ARRAY[1..100] OF BOOL;
	myUsrLive:ARRAY[1..100] OF TP;
	myUserTrigger:ARRAY[1..100] OF F_TRIG;
	
	UsrInList: BOOL;
	test: INT;
	sLogOutString: STRING;
	myDT: DATE_AND_TIME;
	sDT: STRING;
	sLogInString: STRING(255);
	
	sLogInStringOld: STRING;
	xSetLoginTx: BOOL;
	sLogOutStringOld: STRING;
	xSetLogOutTx: BOOL;
	
	myUserName: WSTRING;
END_VAR


myUserName:=VisuElems.CurrentFullUserName;
myUsrName:=WSTRING_TO_STRING(myUserName);


IF myUsrName<>'' THEN
		
	
	UsrInList:=FALSE;
	FOR i:=1 TO 100 DO
		IF myUsrName=UserList[i] THEN // UsrName in List
			UsrIdxLive[i]:=TRUE;
			UsrInList:=TRUE;
		ELSE
			UsrIdxLive[i]:=FALSE;
			test:=test+1;
			
		END_IF
		
		myUsrLive[i](IN:=UsrIdxLive[i] , PT:=T#60S  ); //Extending UsrEntry for another 60s
		myUserTrigger[i](CLK:=myUsrLive[i].Q  );
		
		IF myUserTrigger[i].Q THEN // deleting Entry after 60 s
			myDT:=FuGetDateAndTime();
			sDT:=DT_TO_STRING(myDT);
			sLogOutString:=CONCAT('LogOut: ',UserList[i]);
			sLogOutString:=CONCAT(sLogOutString,',');
			sLogOutString:=CONCAT(sLogOutString,sDT);
			UserList[i]:='';
			
		END_IF
		
			
	END_FOR
	
	
	IF NOT UsrInList THEN //User Not in List
		FOR i:=1 TO 100 DO
			IF UserList[i]='' AND NOT UsrInList THEN //search for the next free entry
				UserList[i]:=myUsrName;
				UsrInList:=TRUE;
					myDT:=FuGetDateAndTime();
					sDT:=DT_TO_STRING(myDT);
					sLogInString:=CONCAT('LogIn: ',UserList[i]);
					sLogInString:=CONCAT(sLogInString,',');
					sLogInString:=CONCAT(sLogInString,sDT);
				EXIT;
			END_IF
		END_FOR
	END_IF
END_IF


IF sLogInString<>sLogInStringOld THEN
	xSetLoginTx:=TRUE;
	sLogInStringOld:=sLogInString;
END_IF
IF sLogOutString<>sLogOutStringOld THEN
	xSetLogOutTx:=TRUE;
	sLogOutStringOld:=sLogOutString;
END_IF

END_FUNCTION_BLOCK

// 30 Visualizations/DynVisuElems/building/sunblind01/sunblind01Visu
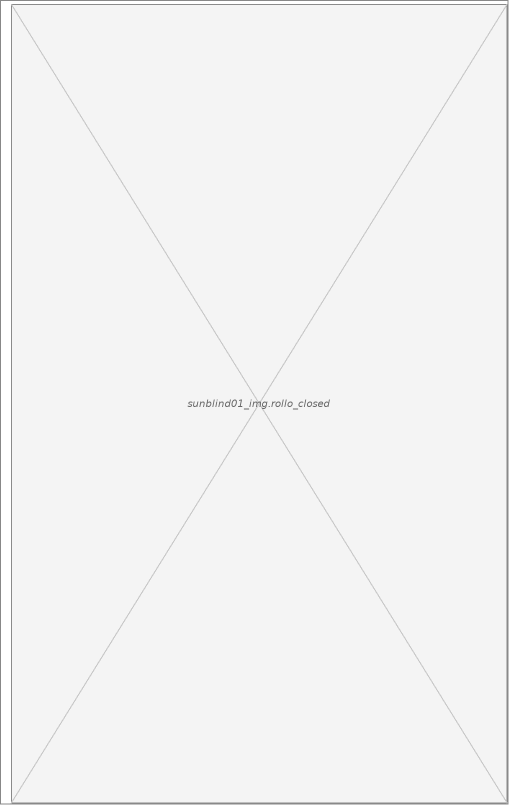
VISUALIZATION sunblind01Visu  // 509x805
VAR_IN_OUT
	sID:STRING;
END_VAR
    Image (11,4 496x799), image: sunblind01_img.rollo_closed
        p84334746: sID
END_VISUALIZATION

// 30 Visualizations/DynVisuElems/cogwheels/cogwheel01/cogwheel01Visu
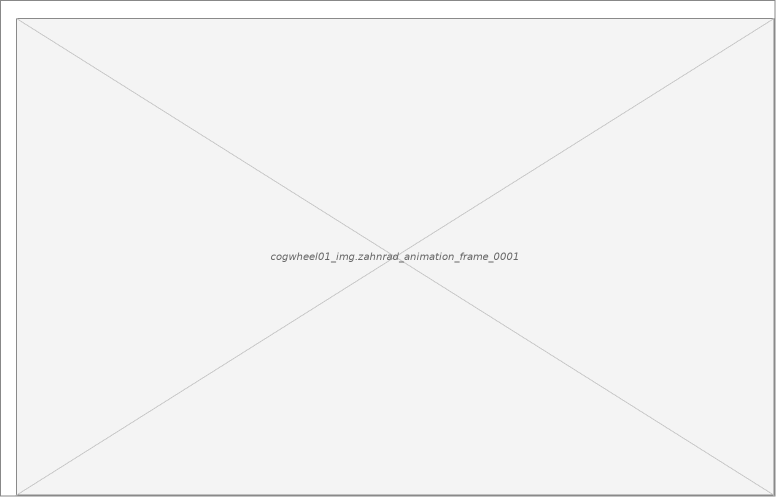
VISUALIZATION cogwheel01Visu  // 776x497
VAR_IN_OUT
	sID:STRING;
END_VAR
    Image (16,18 758x477), image: cogwheel01_img.zahnrad_animation_frame_0001
        p84334746: sID
END_VISUALIZATION

// 30 Visualizations/DynVisuElems/cogwheels/cogwheel02/cogwheel02Visu
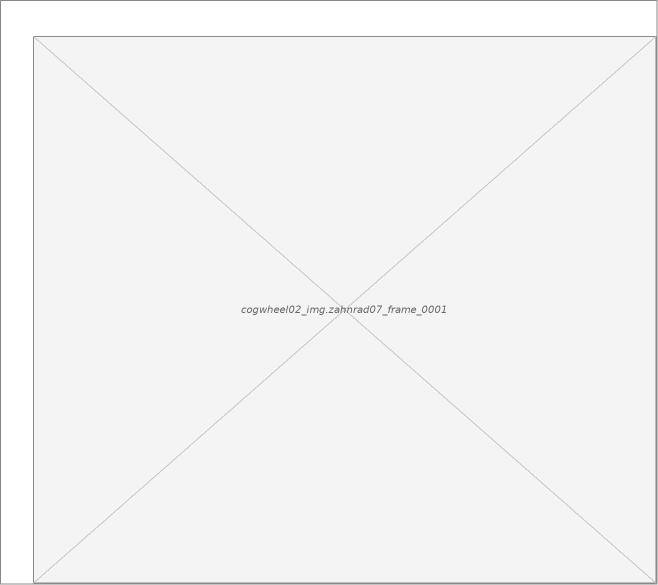
VISUALIZATION cogwheel02Visu  // 658x585
VAR_IN_OUT
	sID:STRING;
END_VAR
    Image (33,36 623x547), image: cogwheel02_img.zahnrad07_frame_0001
        p84334746: sID
END_VISUALIZATION

// 30 Visualizations/DynVisuElems/cogwheels/cogwheel03/cogwheel03Visu
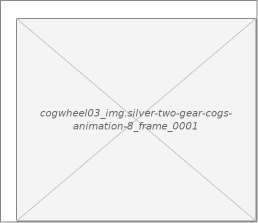
VISUALIZATION cogwheel03Visu  // 258x223
VAR_IN_OUT
	sID:STRING;
END_VAR
    Image (16,18 240x203), image: cogwheel03_img.silver-two-gear-cogs-animation-8_frame_0001
        p84334746: sID
END_VISUALIZATION
